        -0.021266481483774708,0.0,0.0,1.0,0.0,0.0,0.0,0.0,0.0,-0.0,-0.0,-1.0,-0.0,-0.0,-0.0,0.00058545213764139327,
        0.00069492775754933231,-0.013354826750081004,-0.015696387656065527,-0.016360391103343891,
        -0.0004481686028084641,0.013354826750081004,0.015696387656065527,0.016360391103343894,0.0,0.0,1.0,0.0,0.0,
        0.0,0.0,0.0,-0.0,-0.0,-1.0,-0.0,-0.0,-0.0,0.00070855886012245251,0.0163604987338591,-0.010053959431077385,
        -0.013815029502340643,-0.00070322802658466608,0.0,0.0,1.0,0.0,0.0,0.0,0.0,0.0,-0.0,-0.0,-1.0,-0.0,-0.0,-0.0,
        -0.0,0.00066290338327761684,0.00063267402481259919,-0.016360399418003064,0.013354829801521528,
        0.0156963952424949,0.016360399418003064,0.0,0.0,1.0,0.0,0.0,0.0,0.0,0.0,0.0,0.0,-0.0,-0.0,-1.0,-0.0,-0.0,
        -0.0,-0.0,0.00070871228093573281,-0.013354886628180915,-0.00070338839082327207,0.019136254043089867,
        0.019674776790317688,0.0,0.0,1.0,0.0,0.0,0.0,0.0,0.0,-0.0,-0.0,-1.0,-0.0,-0.0,-0.0,-0.0,-0.0,
        0.00070977892002071054,-0.015696489327294644,-0.00070486724956031889,0.0078498358546025652,
        0.021266597087506126,0.0,0.0,1.0,0.0,0.0,0.0,0.0,-0.0,-0.0,-1.0,-0.0,-0.0,-0.0,-0.0,0.00070855886012245251,
        -0.016360498733859103,-0.00070322802658466608,-0.00064115033886434007,0.010053959431077382,
        0.013815029502340643,0.0,0.0,1.0,0.0,0.0,0.0,0.0,-0.0,-0.0,-1.0,-0.0,-0.0,-0.0,-0.0,-0.0,
        0.015696429274739486,0.0007402725668637,0.013814978346247547,0.00078483961287594765,-0.0078505504957846264,
        -0.00059026517985183739,0.0,0.0,1.0,0.0,0.0,0.0,0.0,0.0,-0.0,-0.0,-1.0,-0.0,-0.0,-0.0,0.015696496781502492,
        0.00072094437214855291,0.013815028737181446,-0.0078505344125935073,-0.00078505003013483422,0.0,0.0,1.0,0.0,
        0.0,0.0,0.0,0.0,-0.0,-0.0,-1.0,-0.0,-0.0,-0.0,0.015696489327294647,0.00064281278721221359,
        0.013815029502340637,-0.0007099847981285385,-0.00785055587835492,0.00070514735512079252,0.0,0.0,1.0,0.0,0.0,
        0.0,0.0,0.0,-0.0,-0.0,-1.0,-0.0,-0.0,-0.0,-0.0,0.013814978346247547,-0.000740509959887708,
        -0.0078505513076336172,0.0005902592207076454,0.00045900348534280938,0.0,0.0,1.0,0.0,0.0,-0.0,-1.0,-0.0,-0.0,
        -0.0,0.00073887229766321256,0.016360436265260729,0.00078356528008410354,-0.00058935731463155463,
        -0.013814967279330388,0.0,0.0,1.0,0.0,0.0,0.0,0.0,0.0,-0.0,-0.0,-1.0,-0.0,-0.0,-0.0,0.00073903425520360994,
        0.019674701485866784,0.00078374994311404967,-0.01335483887448634,-0.00058948103625439357,
        0.019136152968431349,0.0,0.0,1.0,0.0,0.0,0.0,0.0,0.0,-0.0,-0.0,-1.0,-0.0,-0.0,-0.0,-0.0,
        0.0007402725668636999,0.00078483961287594722,-0.015696416044310803,-0.00059013581334217832,
        0.0078498304624371844,0.021266532224969138,0.0,0.0,0.0,0.0,0.0,-0.0,-1.0,-0.0,-0.0,-0.0,
        0.00073887229766321256,0.01005394241171902,0.01381497834624754,0.00078356528008410354,-0.016360422411734073,
        -0.00058935731463155463,0.0,0.0,1.0,0.0,0.0,0.0,0.0,-0.0,-0.0,-1.0,-0.0,-0.0,-0.0,-0.0,0.016360509090127547,
        0.00071950068311493818,-0.013815028737181451,-0.00078356528008410376,0.0,0.0,1.0,0.0,0.0,0.0,0.0,0.0,-0.0,
        -0.0,-1.0,-0.0,-0.0,-0.0,0.0163604987338591,-0.0007085588601224524,-0.013815029502340658,
        0.00070322802658466575,0.00064115033886434007,0.0,0.0,1.0,0.0,0.0,0.0,0.0,0.0,-0.0,-0.0,-1.0,-0.0,-0.0,-0.0,
        -0.0,0.016360436265260726,-0.00073887229766321266,-0.013814978346247555,0.00058935142225332476,
        0.00045695607481956147,0.0,0.0,1.0,0.0,0.0,-0.0,-1.0,-0.0,-0.0,-0.0,0.016360509090127547,
        -0.00071950068311493818,-0.010053942472644632,-0.013815028737181451,0.00066772991164514863,
        0.00078356528008410376,0.0,0.0,1.0,0.0,0.0,0.0,0.0,-0.0,-0.0,-1.0,-0.0,-0.0,-0.0,-0.0,
        0.00071965353685171413,-0.013354881724508197,-0.00078374994311405011,0.01913627908650653,
        0.019674802040209546,0.0,0.0,1.0,0.0,0.0,0.0,0.0,0.0,-0.0,-0.0,-1.0,-0.0,-0.0,-0.0,-0.0,
        0.00072094437214855281,-0.015696496781502488,-0.00078483961287594754,0.0078498143875897573,
        0.021266622548422189,0.0,0.0,0.0,0.0,0.0,-0.0,-1.0,-0.0,-0.0,-0.0,0.00071950068311493818,
        -0.016360509090127547,-0.00078356528008410376,0.010053942472644628,0.013815028737181455,0.0,0.0,1.0,0.0,0.0,
        0.0,0.0,-0.0,-0.0,-1.0,-0.0,-0.0,-0.0,-0.0,-0.013354886628180915,-0.00070871228093573313,
        0.019136254043089853,0.00070338839082327153,0.019674776790317681,0.00064128274259411333,0.0,0.0,1.0,0.0,0.0,
        0.0,0.0,0.0,-0.0,-0.0,-1.0,-0.0,-0.0,-0.0,-0.0,-0.0,-0.0078497740839998265,-0.01913681977138957,
        -0.00071047308705639756,0.021264803951796803,0.00072175936181417908,0.0,0.0,1.0,0.0,0.0,0.0,0.0,-0.0,-0.0,
        -1.0,-0.0,-0.0,-0.0,-0.0,-0.0,-0.013354847416887408,-0.00073903425520361,0.00058947514464916862,
        0.019136171450666897,0.019674701485866791,0.00045700543323026538,0.0,0.0,1.0,0.0,0.0,-0.0,-1.0,-0.0,-0.0,
        -0.0,-0.0,-0.010053984761327205,-0.019675305114254357,-0.0078504940691149945,-0.021264803951796817,
        -0.00071067908889347979,-0.00074130273940990277,-0.00072200639376403209,0.00071067908889347979,
        0.00072200639376403209,0.0,0.0,1.0,0.0,0.0,0.0,0.0,0.0,-0.0,-0.0,-1.0,-0.0,-0.0,-0.0,-0.0,-0.0,-0.0,
        -0.013354881724508197,-0.00071965353685171413,0.00066787723649602772,0.01913627908650652,
        0.00078374994311405,0.019674802040209542,0.0,0.0,1.0,0.0,0.0,0.0,0.0,-0.0,-0.0,-1.0,-0.0,-0.0,-0.0,-0.0,
        -0.0,-0.00070977892002071054,-0.015696489327294644,0.0078498358546025652,0.00070486724956031889,
        0.021266597087506126,0.00064281278721221337,0.0,0.0,0.0,0.0,0.0,-0.0,-1.0,-0.0,-0.0,-0.0,-0.0,
        -0.00058545213764139327,-0.00069492775754933231,-0.013354826750081004,-0.015696387656065527,
        -0.016360391103343891,0.013354826750081004,0.015696387656065527,0.016360391103343894,0.0004481686028084641,
        0.0,0.0,1.0,0.0,0.0,0.0,-0.0,-0.0,-1.0,-0.0,-0.0,-0.0,-0.0,-0.0,-0.00070855886012245251,
        -0.016360498733859103,0.010053959431077382,0.013815029502340643,0.00070322802658466608,
        0.00064115033886434007,0.0,0.0,1.0,0.0,0.0,0.0,0.0,-0.0,-0.0,-1.0,-0.0,-0.0,-0.0,-0.0,-0.0,
        -0.00066290338327761684,-0.00063267402481259919,-0.016360399418003064,0.013354829801521528,
        0.00082020698923774085,0.0,0.0,1.0,0.0,0.0,0.0,0.0,-0.0,-0.0,-1.0,-0.0,-0.0,-0.0,-0.0,-0.015696429274739486,
        -0.0007402725668637,0.0078498312759191675,0.0005901298647647122,0.021266544761989165,0.00045868723263609631,
        0.0,0.0,0.0,0.0,-1.0,-0.0,-0.0,-0.0,-0.015696496781502492,-0.013815028737181443,-0.00072119125834864851,
        0.0078505344125935142,0.00066885432718430675,0.00078505003013483422,0.0,0.0,1.0,0.0,0.0,0.0,-0.0,-0.0,-1.0,
        -0.0,-0.0,-0.0,-0.0,-0.0,-0.00073887229766321256,-0.016360436265260733,0.01005394241171902,
        0.00058935142225332476,0.013814978346247547,0.00045695607481956217,0.0,0.0,1.0,0.0,0.0,0.0,-0.0,-0.0,-1.0,
        -0.0,-0.0,-0.0,-0.0,-0.01636050909012755,-0.00071950068311493818,0.010053942472644628,
        0.00066772991164514863,0.01381502873718145,0.00078356528008410376,0.0,0.0,1.0,0.0,0.0,0.0,-0.0,-0.0,-1.0,
        -0.0,-0.0,-0.0,-0.0,-0.0,0.019136104037587275,0.0078505627081109745,0.00059070966910656456,
        4.6667541046249082E-6,-0.00046016924547736962,0.0,0.0,1.0,0.0,0.0,0.0,0.0,0.0,0.0,-0.0,-0.0,-1.0,-0.0,-0.0,
        -0.0,0.013354826750081004,0.000589475144649169,0.00070338839082327109,-0.019136104037587275,
        -0.00045721508909140403,0.0,0.0,1.0,0.0,0.0,0.0,-0.0,-1.0,-0.0,-0.0,-0.0,-0.0,0.01005395943107738,
        0.019674776790317691,0.0078505558783549187,0.00071067908889347968,-0.00070606688480528491,0.0,0.0,1.0,0.0,
        0.0,0.0,0.0,0.0,0.0,-0.0,-0.0,-1.0,-0.0,-0.0,-0.0,-0.0,0.01335483887448634,-0.00058948103625439325,-0.0,
        0.00045964338544026849,0.0078505504957846264,7.1576985742576626E-6,1.0242094517058181E-6,0.0,0.0,1.0,0.0,
        0.0,0.0,0.0,0.0,0.0,-0.0,-0.0,-1.0,-0.0,-0.0,-0.0,0.010053942472644626,0.019674802040209546,
        0.007850534412593509,0.021264422151952962,-0.00072200639376403209,0.00066940907433716364,
        0.00078577738649557045,0.0,0.0,1.0,0.0,0.0,0.0,0.0,0.0,-0.0,-0.0,-1.0,-0.0,-0.0,-0.0,-0.0,
        0.013354826750081004,-0.000589475144649169,-0.00070338839082327109,-0.019136104037587275,
        0.00045721508909140403,0.0,0.0,1.0,0.0,0.0,0.0,-0.0,-0.0,-1.0,-0.0,-0.0,-0.0,-0.0,-0.0,0.01335483887448634,
        -0.00078374994311405,-0.019136152968431349,-0.019674684401114268,0.00058948103625439325,0.0,0.0,1.0,0.0,0.0,
        0.0,0.0,-0.0,-0.0,-1.0,-0.0,-0.0,-0.0,-0.0,-0.0,0.00070998479812853861,0.013815029502340646,
        0.021266597087506119,-0.007850555878354917,-0.000705147355120792,0.0,0.0,1.0,0.0,0.0,0.0,0.0,0.0,-0.0,-0.0,
        -1.0,-0.0,-0.0,-0.0,-0.0,0.0007032280265846663,0.016360391103343884,0.000589357314631555,
        -0.013814936811065831,0.0,0.0,1.0,0.0,0.0,0.0,0.0,0.0,0.0,-0.0,-0.0,-1.0,-0.0,-0.0,-0.0,
        0.00058545773453366594,9.9821594966206443E-7,-0.013354818196216901,-0.015696374407663447,
        -0.016360377230620737,0.013354818196216901,0.015696374407663447,0.016360377230620737,0.0,0.0,1.0,0.0,0.0,
        0.0,0.0,0.0,0.0,0.0,-0.0,-0.0,-1.0,-0.0,-0.0,-0.0,-0.0,0.00070338839082327185,0.019674637958108528,
        0.00058948103625439336,-0.013354818196216903,0.019136085528464446,0.0,0.0,1.0,0.0,0.0,0.0,0.0,0.0,0.0,-0.0,
        -0.0,-1.0,-0.0,-0.0,-0.0,-0.0,0.0007048672495603191,0.00059013581334217821,-0.015696374407663444,
        0.00784984185776794,0.021266481483774712,0.0,0.0,0.0,0.0,0.0,0.0,-0.0,-1.0,-0.0,-0.0,-0.0,
        0.00058935142225332465,0.0007032280265846663,-0.016360391103343887,-0.0004571656718651675,
        0.010053943283910695,0.013814947892318402,0.0,0.0,1.0,0.0,0.0,0.0,0.0,-0.0,-0.0,-1.0,-0.0,-0.0,-0.0,
        0.00058935731463155485,1.0183040766464289E-6,-0.00013071479116047661,0.010053939720042822,
        0.013814936811065836,0.0,0.0,1.0,0.0,0.0,0.0,0.0,0.0,-0.0,-0.0,-1.0,-0.0,-0.0,-0.0,-0.0,
        0.00071047308705639756,-0.0078498358546025635,-0.019136254043089867,0.021264396690767625,0.0,0.0,1.0,0.0,
        0.0,0.0,0.0,-0.0,-0.0,-1.0,-0.0,-0.0,-0.0,-0.0,-0.0,0.00071029983670461863,0.00059047175686875969,
        -0.010053943283910698,-0.019674637958108521,-0.00045960759224737192,0.01804924706676608,0.0,1.0,0.0,0.0,0.0,
        0.0,-0.0,-0.0,-1.0,-0.0,-0.0,-0.0,-0.0,0.00070998479812853861,-0.013815029502340641,-0.000705147355120792,
        -0.00064310201354924451,0.007850555878354917,0.0,0.0,1.0,0.0,0.0,0.0,0.0,-0.0,-0.0,-1.0,-0.0,-0.0,-0.0,-0.0,
        -0.0,0.013815028737181446,0.021266622548422178,-0.00072119125834864851,-0.0078505344125935073,
        0.00066885432718430675,0.00078505003013483422,0.0,0.0,1.0,0.0,0.0,0.0,0.0,-0.0,-0.0,-1.0,-0.0,-0.0,-0.0,
        -0.0,0.013814947892318402,-0.0005902592207076454,-0.00070514735512079263,-0.0078505627081109815,
        0.00045921295820314543,0.0,0.0,1.0,0.0,0.0,-1.0,-0.0,-0.0,-0.0,-0.0,-0.0,0.015696416044310803,
        0.01381496727933039,-0.00078505003013483454,-0.0078505504957846247,0.00059026517985183728,0.0,0.0,1.0,0.0,
        0.0,0.0,0.0,-0.0,-0.0,-1.0,-0.0,-0.0,-0.0,-0.0,0.0007408652531395556,-0.010053942411719023,
        -0.019674701485866784,-0.00059047175686875969,-0.00045939812049741193,0.018049321508312247,0.0,1.0,0.0,0.0,
        0.0,-0.0,-0.0,-1.0,-0.0,-0.0,-0.0,-0.0,0.00074050995988770782,0.00078505003013483476,-0.013814967279330386,
        -0.00059026517985183717,0.007850550495784623,0.0,0.0,1.0,0.0,0.0,0.0,0.0,-0.0,-0.0,-1.0,-0.0,-0.0,-0.0,-0.0,
        0.016360391103343887,-0.00058935142225332465,-0.000703228026584666,-0.013814947892318404,
        0.00045716567186516885,0.0,0.0,1.0,0.0,0.0,-1.0,-0.0,-0.0,-0.0,-0.0,-0.0,-0.00066772991164514874,
        -0.00064115033886434018,-0.01381495313599773,0.00013071479116047655,-0.00058935731463155463,
        -0.010053939720042825,0.0,0.0,1.0,0.0,0.0,0.0,0.0,-0.0,-0.0,-1.0,-0.0,-0.0,-0.0,-0.0,-0.0,
        0.016360422411734077,-0.00078356528008410322,-0.010053938852608935,-0.013814967279330383,
        0.00058935731463155474,0.0,0.0,1.0,0.0,0.0,0.0,0.0,-0.0,-0.0,-1.0,-0.0,-0.0,-0.0,-0.0,
        0.00072155339410677672,-0.010053942472644626,-0.019674802040209542,-0.00078538438365502385,
        0.018049442230007151,0.0,0.0,1.0,0.0,0.0,0.0,0.0,-0.0,-0.0,-1.0,-0.0,-0.0,-0.0,-0.0,0.0007211912583486484,
        -0.01381502873718145,-0.00078505003013483443,0.0078505344125935073,0.0,0.0,1.0,0.0,0.0,0.0,0.0,-0.0,-0.0,
        -1.0,-0.0,-0.0,-0.0,-0.0,-0.010053959431077376,-0.00071029983670461863,-0.019674776790317688,
        -0.0078505558783549187,0.00070606688480528491,0.00064403085718071711,0.0,0.0,1.0,0.0,0.0,0.0,0.0,-0.0,-0.0,
        -1.0,-0.0,-0.0,-0.0,-0.0,-0.0,-0.0,-0.013354829801521528,-0.00066787723649602794,-0.00064128274259411312,
        0.019136117134310814,0.00082836908801823649,0.019674650101301497,0.0,1.0,0.0,0.0,0.0,0.0,-0.0,-0.0,-1.0,
        -0.0,-0.0,-0.0,-0.0,-0.0,-0.019136279086506527,-0.0078505344125935073,-0.018049442230007113,
        -0.00072200639376403209,0.00078577738649557045,0.0,0.0,1.0,0.0,0.0,0.0,-0.0,-0.0,-1.0,-0.0,-0.0,-0.0,-0.0,
        -0.0,-0.0,-0.010053942411719021,-0.0007408652531395556,-0.019674701485866787,0.00059047175686876,
        0.018049321508312247,0.00045939812049741166,0.0,1.0,0.0,0.0,-0.0,-1.0,-0.0,-0.0,-0.0,-0.0,
        -0.01335483887448634,-0.00078374994311405,0.00058948103625439325,0.019136152968431349,0.019674684401114268,
        0.0,0.0,1.0,0.0,0.0,0.0,0.0,-0.0,-0.0,-1.0,-0.0,-0.0,-0.0,-0.0,-0.0,-0.010053942472644626,
        -0.019674802040209546,-0.00072155339410677683,0.00066911306678242447,0.018049442230007123,
        0.00078538438365502352,0.0,1.0,0.0,0.0,0.0,-0.0,-0.0,-1.0,-0.0,-0.0,-0.0,-0.0,-0.00070998479812853861,
        -0.013815029502340641,0.007850555878354917,0.000705147355120792,0.00064310201354924451,0.0,0.0,1.0,0.0,0.0,
        0.0,0.0,-0.0,-0.0,-1.0,-0.0,-0.0,-0.0,-0.0,-0.0,-0.00066869452258176915,-0.015696395242494905,
        -0.00064281278721221348,0.0078498388863461367,0.00082974490333613884,0.021266503270189141,0.0,0.0,0.0,0.0,
        -0.0,-1.0,-0.0,-0.0,-0.0,-0.0,-0.00058545773453366594,-3.5950544673529394E-6,-0.013354818196216901,
        -0.015696374407663447,-0.016360377230620737,0.013354818196216901,0.015696374407663447,0.016360377230620737,
        0.0,0.0,1.0,0.0,0.0,0.0,0.0,0.0,-0.0,-0.0,-1.0,-0.0,-0.0,-0.0,-0.0,-0.0,-0.0,-0.013814978346247541,
        -0.00074050995988770782,0.0078505513076336225,0.00059025922070764572,0.00045900348534281133,0.0,0.0,1.0,0.0,
        0.0,0.0,-0.0,-0.0,-1.0,-0.0,-0.0,-0.0,-0.0,-0.015696416044310803,-0.00078483961287594765,
        0.0078498304624371948,0.00059013581334217821,0.021266532224969107,0.0,0.0,1.0,0.0,0.0,0.0,-0.0,-0.0,-1.0,
        -0.0,-0.0,-0.0,-0.0,-0.00078356528008410354,-0.016360422411734073,0.010053938852608933,
        0.00058935731463155463,0.013814967279330381,0.0,0.0,1.0,0.0,0.0,0.0,-0.0,-0.0,-1.0,-0.0,-0.0,-0.0,-0.0,-0.0,
        0.013354818196216903,0.00058948103625439347,0.0004572150890914036,-0.01913608552846445,0.0,0.0,1.0,0.0,0.0,
        0.0,0.0,0.0,0.0,-0.0,-0.0,-1.0,-0.0,-0.0,-0.0,-0.0,0.007850555878354917,4.72166684662135E-5,
        -0.00071067908889347968,0.00070606688480528491,0.00064403085718071711,0.0,0.0,1.0,0.0,0.0,0.0,0.0,0.0,0.0,
        -0.0,-0.0,-1.0,-0.0,-0.0,-0.0,-0.0,0.0078505513076336155,0.021264344306911508,-0.00074130273940990277,
        0.00059070966910656445,0.00045995981458200994,0.0,0.0,1.0,0.0,0.0,0.0,-0.0,-1.0,-0.0,-0.0,-0.0,
        0.019136104037587285,-0.00070578661505656148,0.0078505627081109728,-0.00059070966910656456,
        -4.6667541046249082E-6,0.00046016924547737027,0.0,0.0,1.0,0.0,0.0,-1.0,-0.0,-0.0,-0.0,-0.0,-0.0,
        0.010053938852608935,0.019674684401114268,-0.00078538438365502331,0.0078505504957846282,
        -7.1576985742576693E-6,0.00059071565881779026,0.0,0.0,1.0,0.0,0.0,0.0,0.0,0.0,-0.0,-0.0,-1.0,-0.0,-0.0,-0.0,
        -0.0,0.013354818196216903,-0.00058948103625439347,-0.00082836908801823736,-0.01913608552846445,
        -0.019674620847241392,0.0,0.0,1.0,0.0,0.0,0.0,0.0,-0.0,-0.0,-1.0,-0.0,-0.0,-0.0,-0.0,-0.0,-0.0,
        0.0078498304624371861,0.019136152968431349,-0.00078556684097776574,-0.021264331757721504,
        0.00059058621231803418,0.0,0.0,1.0,0.0,0.0,0.0,0.0,-0.0,-0.0,-1.0,-0.0,-0.0,-0.0,0.013814947892318409,
        0.0007051473551207923,0.0212664940442422,0.0005902651798518375,4.7206293852370952E-5,-0.007850561894963819,
        0.0,0.0,1.0,0.0,0.0,0.0,0.0,0.0,0.0,-0.0,-0.0,-1.0,-0.0,-0.0,-0.0,0.00059025922070764572,
        0.00070514735512079241,-0.013814947892318418,-0.00045921295820314608,0.0078505627081109711,0.0,0.0,1.0,0.0,
        0.0,0.0,0.0,-0.0,-0.0,-1.0,-0.0,-0.0,-0.0,1.0250173309722677E-6,0.0,-0.0,0.00059070966910656467,
        -0.0078505627081109745,-7.8752164488168983E-5,0.0,0.0,1.0,0.0,0.0,0.0,0.0,-0.0,-0.0,-1.0,-0.0,-0.0,-0.0,
        -0.0,0.00059026517985183772,1.0228783844071197E-6,-0.00012539822612430226,0.0078505618949638225,0.0,0.0,1.0,
        0.0,0.0,0.0,0.0,0.0,-0.0,-0.0,-1.0,-0.0,-0.0,-0.0,-0.0,0.00071067908889347979,-0.0078505558783549152,
        -7.8751758300344045E-5,-0.00070606688480528469,-0.00064403085718071711,0.0,0.0,1.0,0.0,0.0,0.0,0.0,-0.0,
        -0.0,-1.0,-0.0,-0.0,-0.0,-0.0,-0.0,-0.0,-0.00066885432718430643,-0.000643102013549245,-0.0078505589212312,
        0.00012539822612430221,-0.00059026517985183706,0.0,0.0,1.0,0.0,0.0,0.0,0.0,-0.0,-0.0,-1.0,-0.0,-0.0,-0.0,
        -0.0,-0.0,0.00045939812049741,-0.010053938852608933,-0.019674684401114268,-0.00059047772800183325,
        7.1576985742576753E-6,1.0242094517058098E-6,-0.00785055049578463,0.0,0.0,1.0,0.0,0.0,0.0,0.0,-0.0,-0.0,-1.0,
        -0.0,-0.0,-0.0,-0.0,-0.0,0.00074130273940990277,-0.00785055130763362,-0.018049321508312233,
        -0.00059070966910656445,-0.00045995981458201091,0.0,0.0,1.0,0.0,0.0,0.0,-0.0,-0.0,-1.0,-0.0,-0.0,-0.0,-0.0,
        -0.0,0.00072200639376403209,-0.007850534412593509,-0.018049442230007113,-0.00078577738649557056,0.0,0.0,1.0,
        0.0,0.0,0.0,0.0,-0.0,-0.0,-1.0,-0.0,-0.0,-0.0,-0.0,-0.0,-0.010053941700689279,-0.00066911306678242458,
        -0.019674650101301497,-0.00064350274257291972,0.018049261985986123,0.00083041340795978814,1.0,0.0,0.0,0.0,
        -0.0,-0.0,-1.0,-0.0,-0.0,-0.0,-0.0,-0.0,-0.013354818196216903,-0.00058948103625439347,
        -0.00082836908801823736,0.01913608552846445,0.019674620847241395,0.0,0.0,1.0,0.0,0.0,0.0,0.0,-0.0,-0.0,-1.0,
        -0.0,-0.0,-0.0,-0.0,-0.0,-0.0,-0.00074130273940990277,-0.0,-0.0078498304624371861,-0.019136152968431349,
        -0.00078556684097776574,0.00059058621231803418,0.0,0.0,1.0,0.0,0.0,0.0,-0.0,-0.0,-1.0,-0.0,-0.0,-0.0,-0.0,
        -0.0,-0.010053938852608928,-0.00078538438365502374,-0.019674684401114275,0.00059047772800183335,
        0.018049300450950378,0.0,1.0,0.0,0.0,0.0,-0.0,-0.0,-1.0,-0.0,-0.0,-0.0,-0.0,-0.015696374407663447,
        -0.0005902651798518375,-0.00012539822612430229,-1.0228783844071214E-6,0.007850561894963819,0.0,0.0,1.0,0.0,
        0.0,0.0,-0.0,-0.0,-1.0,-0.0,-0.0,-0.0,-0.0,-0.0,-0.0,-0.000589357314631555,-3.6300677219671527E-6,
        -0.00013071479116047663,0.01005393972004282,0.013814936811065819,0.0,0.0,1.0,0.0,0.0,0.0,-0.0,-0.0,-1.0,
        -0.0,-0.0,-0.0,-0.0,-0.0,-0.0,-0.013814967279330381,-0.00078505003013483476,-0.021266532224969107,
        -0.00045900348534281117,0.0078505504957846247,0.00059026517985183739,0.0,0.0,1.0,0.0,0.0,0.0,-0.0,-0.0,-1.0,
        -0.0,-0.0,-0.0,-0.0,-0.0,0.0078498418577679363,0.00059058621231803429,0.00012594643379194981,
        1.0243116170212105E-6,-0.021264280982048623,0.0,0.0,1.0,0.0,0.0,0.0,0.0,0.0,0.0,-0.0,-0.0,-1.0,-0.0,-0.0,
        -0.0,0.007850558921231196,-2.8452679316136533E-6,0.0008309073466565292,0.0,0.0,1.0,0.0,0.0,0.0,0.0,0.0,0.0,
        -0.0,-0.0,-1.0,-0.0,-0.0,-0.0,-0.0,0.0078498418577679328,-3.6410799041126835E-6,7.8752197135979057E-5,
        -0.00059071565881779048,-3.6422315821786528E-6,0.0,0.0,1.0,0.0,0.0,0.0,0.0,0.0,-0.0,-0.0,-1.0,-0.0,-0.0,
        -0.0,-0.0,-0.0,0.01005393972004282,8.6574413715050772E-5,-0.00059047772800183325,-0.018049225981178776,0.0,
        0.0,1.0,0.0,0.0,0.0,0.0,-0.0,-0.0,-1.0,-0.0,-0.0,-0.0,-0.0,-0.0,-0.01005393972004282,
        -0.00059047772800183325,-3.6400546269338619E-6,-8.6574413715050745E-5,0.018049225981178765,0.0,1.0,0.0,0.0,
        0.0,-0.0,-0.0,-1.0,-0.0,-0.0,-0.0,-0.0,-0.0,-0.0078498418577679363,-0.00012594643379194981,
        -0.00059071565881779048,-1.0250173309722696E-6,0.0,0.0,1.0,0.0,0.0,0.0,-0.0,-0.0,-1.0,-0.0,-0.0,-0.0,-0.0,
        -0.0,-0.0,-0.0,0.00785056189496382,0.00059071565881779048,4.721686715653703E-5,1.0250173309722696E-6,0.0,
        0.0,1.0,0.0,0.0,0.0,0.0,0.0,0.0,0.0,-0.0,-0.0,-1.0,-0.0,-0.0,-0.0,-0.002139599215214946,
        -0.023117048152407872,-0.0022397649528431126,-0.027072995129471072,-0.0021836277363616002,
        -0.028166145144496873,0.002139599215214946,0.023117048152407872,0.0022397649528431126,0.027072995129471072,
        0.0021836277363616007,0.028166145144496869,0.0,0.0,0.0,1.0,0.0,0.0,0.0,0.0,0.0,0.0,-0.0,-0.0,-0.0,-1.0,-0.0,
        -0.0,-0.0,-0.0,0.0021395992152149455,-0.023117145095115522,-0.0021497242199081533,-0.027072819798329567,
        -0.0019633569630565072,-0.02816590468451018,0.023117145095115522,0.027072819798329567,0.028165904684510173,
        0.0,0.0,0.0,1.0,0.0,0.0,0.0,0.0,0.0,-0.0,-0.0,-0.0,-1.0,-0.0,-0.0,-0.0,-0.0,0.023117048152407872,
        -0.0021505378228925251,-0.0022518711100377505,-0.032822477959688887,-0.00219585787232726,
        -0.0336642766045134,0.0021505378228925251,0.0022518711100377505,0.0021958578723272597,0.0,0.0,0.0,1.0,0.0,
        0.0,0.0,0.0,0.0,-0.0,-0.0,-0.0,-1.0,-0.0,-0.0,-0.0,-0.0,0.0022397649528431126,0.023117136629619534,
        0.028165879272568334,0.002368167038278622,-0.0017636731113387088,-0.023117134816530223,
        -0.027072790466377776,-0.028165871707620763,0.027072790466377776,0.0,0.0,0.0,1.0,0.0,0.0,0.0,0.0,0.0,-0.0,
        -0.0,-0.0,-1.0,-0.0,-0.0,-0.0,0.027072995129471072,0.0021528281310241241,0.0021984476162807444,
        0.023967033731365443,-0.0021532798422932995,-0.013757776970334581,-0.0022549381705200254,
        -0.002198962690806161,0.0,0.0,0.0,1.0,0.0,0.0,0.0,0.0,0.0,-0.0,-0.0,-0.0,-1.0,-0.0,-0.0,-0.0,
        0.0021836277363616002,-0.0020059903769841761,-0.023117107076915992,-0.0023681670382786246,
        -0.027072827080784432,-0.028165923858112191,0.023117107076915992,0.027072827080784432,0.028165923858112184,
        0.0,0.0,0.0,1.0,0.0,0.0,0.0,0.0,0.0,-0.0,-0.0,-0.0,-1.0,-0.0,-0.0,-0.0,0.028166145144496876,
        -0.0021508629271109274,-0.017539733206627071,-0.0022522704855525342,-0.023967033731365443,
        -0.0021962714305260589,0.0021508629271109274,0.0022522704855525342,0.0021962714305260593,0.0,0.0,0.0,1.0,
        0.0,0.0,0.0,0.0,0.0,-0.0,-0.0,-0.0,-1.0,-0.0,-0.0,-0.0,-0.0021395992152149455,-0.023117145095115522,
        -0.027072819798329567,-0.02816590468451018,0.023117145095115522,0.0021497242199081533,0.027072819798329567,
        0.0019633569630565077,0.028165904684510173,0.0,0.0,0.0,1.0,0.0,0.0,0.0,0.0,0.0,-0.0,-0.0,-0.0,-1.0,-0.0,
        -0.0,-0.0,-0.0,-0.023117048152407872,-0.0021505378228925251,-0.0022518711100377505,-0.00219585787232726,
        0.0021505378228925251,0.0022518711100377505,0.032822477959688887,0.0021958578723272597,0.033664276604513384,
        0.0,0.0,0.0,1.0,0.0,0.0,0.0,0.0,0.0,-0.0,-0.0,-0.0,-1.0,-0.0,-0.0,-0.0,-0.0,-0.0022397649528431126,
        -0.0023681670382786225,-0.023117134816530223,-0.027072790466377776,-0.028165871707620763,
        0.0017636731113387079,0.023117134816530223,0.028165871707620756,0.0,0.0,0.0,1.0,0.0,0.0,0.0,0.0,-0.0,-0.0,
        -0.0,-1.0,-0.0,-0.0,-0.0,-0.0,-0.027072995129471072,-0.0021528281310241241,-0.0021984476162807444,
        -0.023967033731365456,-0.0022549381705200254,0.0021532798422932995,0.013757776970334581,
        0.0022549381705200254,0.0021989626908061606,0.0,0.0,0.0,1.0,0.0,0.0,0.0,0.0,-0.0,-0.0,-0.0,-1.0,-0.0,-0.0,
        -0.0,-0.0,-0.0021836277363616007,-0.023117107076915992,-0.027072827080784432,-0.028165923858112191,
        0.0020059903769841761,0.023117107076915992,0.0023681670382786238,0.027072827080784432,0.028165923858112184,
        0.0,0.0,0.0,1.0,0.0,0.0,0.0,0.0,-0.0,-0.0,-0.0,-1.0,-0.0,-0.0,-0.0,-0.0,-0.028166145144496869,
        -0.0021508629271109274,-0.0022522704855525342,-0.0021962714305260589,0.0021508629271109274,
        0.017539733206627078,0.0022522704855525342,0.023967033731365467,0.0021962714305260593,0.0,0.0,0.0,1.0,0.0,
        0.0,0.0,0.0,-0.0,-0.0,-0.0,-1.0,-0.0,-0.0,-0.0,-0.0,0.0021505378228925246,0.023117145095115525,
        -0.0021629274560676956,-0.032821849572960068,-0.0019763195483343526,-0.033663644953626663,0.0,0.0,0.0,1.0,
        0.0,0.0,0.0,0.0,-0.0,-0.0,-0.0,-1.0,-0.0,-0.0,-0.0,-0.0,0.0021497242199081537,0.0017636731113387075,
        0.0025248548165844459,-0.023117153652107741,-0.027072767990336359,-0.028165839066171924,
        0.023117153652107741,0.027072767990336359,0.028165839066171917,0.0,0.0,0.0,1.0,0.0,0.0,0.0,0.0,0.0,0.0,-0.0,
        -0.0,-0.0,-1.0,-0.0,-0.0,-0.0,0.0021528281310241237,-0.013756932403821471,-0.03615897334115932,-0.0,
        0.0017730752489912573,0.027072767990336356,-0.036158836489428262,0.0,0.0,0.0,1.0,0.0,0.0,0.0,0.0,-0.0,-0.0,
        -0.0,-1.0,-0.0,-0.0,0.0020059903769841761,0.0019633569630565068,-0.023117148094275803,
        -0.0025248548165844454,0.028165850749951267,0.0,0.0,0.0,1.0,0.0,0.0,0.0,0.0,-0.0,-0.0,-0.0,-1.0,-0.0,-0.0,
        -0.0,0.0021508629271109274,-0.023967031267238804,-0.0,0.0017716448391260384,0.028165839066171927,0.0,0.0,
        0.0,1.0,0.0,0.0,0.0,0.0,0.0,-0.0,-0.0,-0.0,-1.0,-0.0,-0.0,0.0021505378228925246,-0.023117145095115525,-0.0,
        0.0017714658173675476,-0.0014235573934133095,0.033663511042732373,0.0,0.0,0.0,1.0,0.0,0.0,0.0,0.0,-0.0,-0.0,
        -0.0,-1.0,-0.0,-0.0,-0.0,0.0021528281310241237,-0.027072819798329564,-0.0021657727568646559,
        0.013756932403821471,0.036158973341159265,0.0,0.0,0.0,0.0,0.0,0.0,-0.0,-0.0,-0.0,-1.0,-0.0,-0.0,-0.0,
        0.0021508629271109274,-0.028165904684510176,-0.0021634485653239869,-0.0019768379174131762,
        0.017540054199611115,0.023967031267238814,0.0,0.0,0.0,1.0,0.0,0.0,0.0,-0.0,-0.0,-0.0,-1.0,-0.0,-0.0,-0.0,
        -0.0,0.023117136629619537,0.0022556280308783936,0.013758173064519321,-0.0017741542886565819,
        -0.0014273157197953927,0.0,0.0,0.0,1.0,0.0,0.0,0.0,0.0,-0.0,-0.0,-0.0,-1.0,-0.0,-0.0,0.013756545225322915,
        0.032822477959688887,-0.0021539160439461116,-0.002255628030878394,-0.0021996560033501643,
        -0.036155994182829158,0.0021539160439461116,0.002255628030878394,0.0021996560033501647,0.0,0.0,0.0,1.0,0.0,
        0.0,0.0,0.0,-0.0,-0.0,-0.0,-1.0,-0.0,-0.0,0.023117107076915996,0.0021958578723272597,-0.0020152870120824654,
        -0.0023798449910123255,-0.032821938754042893,0.0,0.0,0.0,1.0,0.0,0.0,0.0,0.0,-0.0,-0.0,-0.0,-1.0,-0.0,-0.0,
        -0.0,0.017539733206627082,0.0336642766045134,-0.00219941213896084,0.00215368729603372,0.0022553827543743792,
        0.00219941213896084,0.0,0.0,0.0,1.0,0.0,0.0,0.0,0.0,0.0,0.0,-0.0,-0.0,-0.0,-1.0,-0.0,-0.0,-0.0,
        0.023117145095115518,-0.0021505378228925251,-0.032821849572960082,0.0021629274560676964,
        0.0019763195483343534,0.0,0.0,0.0,1.0,0.0,0.0,0.0,0.0,-0.0,-0.0,-0.0,-1.0,-0.0,-0.0,-0.0,-0.0,
        0.023117136629619537,-0.00225187111003775,-0.032821807333186945,0.0017714658173675487,0.0014229487589399608,
        0.0,0.0,0.0,1.0,0.0,0.0,0.0,-0.0,-0.0,-0.0,-1.0,-0.0,-0.0,-0.0,0.023117107076915996,-0.0021958578723272597,
        -0.032821938754042893,-0.033663737674327086,0.0020152870120824654,0.0023798449910123263,0.0,0.0,0.0,1.0,0.0,
        0.0,0.0,-0.0,-0.0,-0.0,-1.0,-0.0,-0.0,-0.0,-0.0,0.0022544308843389775,0.027072797014430487,
        0.0023823041653880553,0.023967015852373385,-0.0017733843081747245,-0.013758177150392206,0.0,0.0,0.0,1.0,0.0,
        0.0,0.0,0.0,-0.0,-0.0,-0.0,-1.0,-0.0,-0.0,0.0022522704855525342,0.028165879272568337,0.0023802034757232954,
        -0.0017716448391260397,-0.023967012140249259,0.0,0.0,0.0,1.0,0.0,0.0,0.0,0.0,-0.0,-0.0,-0.0,-1.0,-0.0,-0.0,
        0.0022518711100377505,0.03366360485977575,0.0023798449910123263,-0.023117134816530216,
        -0.0017714855698833817,0.032821793825602318,0.0,0.0,0.0,1.0,0.0,0.0,0.0,0.0,-0.0,-0.0,-0.0,-1.0,-0.0,-0.0,
        -0.0,0.0023823041653880553,-0.027072790466377783,-0.0017730752489912573,0.01375694528625826,
        0.036158931786919049,0.0,0.0,0.0,0.0,0.0,-0.0,-0.0,-1.0,-0.0,-0.0,0.027072827080784432,
        0.0021984476162807444,0.023967007687598831,-0.013758082261467377,-0.0023827866608640042,0.0,0.0,0.0,1.0,0.0,
        0.0,0.0,0.0,-0.0,-0.0,-0.0,-1.0,-0.0,-0.0,0.027072819798329564,0.0019791101348432538,0.0239670312672388,
        -0.0021532798422932995,-0.013758164253474777,0.0021663421034936255,0.0,0.0,0.0,1.0,0.0,0.0,0.0,0.0,-0.0,
        -0.0,-0.0,-1.0,-0.0,-0.0,-0.0,0.02707279701443048,0.023967015852373378,-0.0022549381705200249,
        -0.013758173064519324,0.0017733644650094233,0.001426115796022355,0.0,0.0,1.0,0.0,0.0,-0.0,-0.0,-1.0,-0.0,
        -0.0,0.027072827080784432,0.0020172069825707454,0.0023823041653880544,0.023967007687598831,
        -0.00219896269080616,-0.013758082261467377,0.0,0.0,0.0,1.0,0.0,0.0,0.0,-0.0,-0.0,-0.0,-1.0,-0.0,-0.0,-0.0,
        0.0021962714305260589,0.028165923858112184,-0.0023802034757232967,-0.023967007687598837,0.0,0.0,0.0,1.0,0.0,
        0.0,0.0,0.0,-0.0,-0.0,-0.0,-1.0,-0.0,-0.0,0.0021958578723272597,-0.023117107076915992,
        -0.0023798449910123281,0.032821938754042886,0.033663737674327066,0.0,0.0,0.0,1.0,0.0,0.0,0.0,0.0,-0.0,-0.0,
        -0.0,-1.0,-0.0,-0.0,-0.0,0.002198447616280744,-0.027072827080784435,-0.0023823041653880561,
        0.013756850421972387,0.036159076531973151,0.0,0.0,0.0,0.0,0.0,-0.0,-0.0,-1.0,-0.0,-0.0,
        0.0021962714305260589,-0.028165923858112181,-0.0020155176559669297,-0.0023802034757232967,
        0.017539980122310408,0.023967007687598862,0.0,0.0,0.0,1.0,0.0,0.0,0.0,-0.0,-0.0,-0.0,-1.0,-0.0,-0.0,-0.0,
        0.02816590468451018,-0.0021508629271109274,-0.023967031267238807,0.0021634485653239869,
        0.0019768379174131758,0.0,0.0,0.0,1.0,0.0,0.0,0.0,0.0,-0.0,-0.0,-0.0,-1.0,-0.0,-0.0,-0.0,
        0.028165879272568337,-0.0022522704855525342,-0.023967015852373392,0.0017716250685312594,
        0.0014234593859236441,0.0,0.0,1.0,0.0,0.0,-0.0,-0.0,-1.0,-0.0,-0.0,0.028165923858112191,
        -0.0021962714305260589,-0.023967007687598817,0.0020155176559669297,0.0023802034757232963,0.0,0.0,0.0,1.0,
        0.0,0.0,0.0,-0.0,-0.0,-0.0,-1.0,-0.0,-0.0,-0.0,-0.0021505378228925246,-0.023117145095115525,
        0.0021629274560676956,0.032821849572960068,0.001976319548334353,0.033663644953626656,0.0,0.0,0.0,1.0,0.0,
        0.0,0.0,0.0,-0.0,-0.0,-0.0,-1.0,-0.0,-0.0,-0.0,-0.0,-0.0017636536977724872,-0.0021497242199081537,
        -0.023117155475339022,0.0014113188375514472,0.028165846654428471,0.0,0.0,0.0,1.0,0.0,0.0,0.0,-0.0,-0.0,-0.0,
        -1.0,-0.0,-0.0,-0.0,-0.0,-0.0021528281310241237,-0.027072819798329564,0.013756932403821471,
        0.0021657727568646559,0.0019791101348432556,0.036158973341159265,0.0,0.0,0.0,0.0,0.0,-0.0,-0.0,-1.0,-0.0,
        -0.0,-0.0,-0.0020059903769841757,-0.0019633569630565077,-0.0017636731113387079,-0.0014113188375514463,
        -0.023117153652107741,-0.027072767990336359,-0.028165839066171924,0.023117153652107741,0.028165839066171917,
        0.0,0.0,0.0,1.0,0.0,0.0,0.0,0.0,-0.0,-0.0,-0.0,-1.0,-0.0,-0.0,-0.0,-0.0,-0.0,-0.0021508629271109274,
        -0.028165904684510176,0.017540054199611115,0.0021634485653239869,0.023967031267238814,0.0019768379174131762,
        0.0,0.0,0.0,1.0,0.0,0.0,0.0,-0.0,-0.0,-0.0,-1.0,-0.0,-0.0,-0.0,-0.0,-0.023117136629619537,
        -0.00225187111003775,0.0017714658173675487,0.032821807333186945,0.0014229487589399608,0.033663604859775743,
        0.0,0.0,1.0,0.0,0.0,-0.0,-0.0,-1.0,-0.0,-0.0,-0.0,-0.013756545225322915,-0.032822477959688887,
        -0.0021539160439461116,-0.002255628030878394,-0.0021996560033501643,0.0021539160439461116,
        0.002255628030878394,0.0021996560033501647,0.036155994182829096,0.0,0.0,0.0,0.0,0.0,0.0,-0.0,-0.0,-0.0,-1.0,
        -0.0,-0.0,-0.0,-0.0,-0.023117107076915996,-0.0021958578723272597,0.0020152870120824654,
        0.0023798449910123263,0.032821938754042893,0.033663737674327072,0.0,0.0,0.0,1.0,0.0,0.0,0.0,-0.0,-0.0,-0.0,
        -1.0,-0.0,-0.0,-0.0,-0.0,-0.017539733206627085,-0.033664276604513384,-0.00219941213896084,
        0.00215368729603372,0.03112680478206669,0.0,0.0,0.0,1.0,0.0,0.0,0.0,-0.0,-0.0,-0.0,-1.0,-0.0,-0.0,-0.0,
        -0.0022544308843389775,-0.027072797014430487,0.0017730554216371041,0.013756941202814331,
        0.0014255752842010033,0.0361589433554084,0.0,0.0,0.0,0.0,-0.0,-1.0,-0.0,-0.0,-0.0022522704855525342,
        -0.0023802034757232954,-0.028165871707620752,0.00177164483912604,0.017540060210790732,0.023967012140249284,
        0.0,0.0,0.0,1.0,0.0,0.0,-0.0,-0.0,-0.0,-1.0,-0.0,-0.0,-0.0,-0.0,-0.027072827080784432,
        -0.0021984476162807448,0.0020172069825707454,0.013756850421972387,0.0023823041653880557,
        0.036159076531973207,0.0,0.0,0.0,1.0,0.0,0.0,-0.0,-0.0,-0.0,-1.0,-0.0,-0.0,-0.0,-0.0021962714305260593,
        -0.028165923858112181,0.0020155176559669297,0.017539980122310408,0.0023802034757232963,0.023967007687598862,
        0.0,0.0,0.0,1.0,0.0,0.0,-0.0,-0.0,-0.0,-1.0,-0.0,-0.0,-0.0,-0.0,0.0021670637484648039,0.0017738649457463914,
        0.013757007748269136,0.00021693526799154337,-0.036155235792572543,0.0,0.0,0.0,1.0,0.0,0.0,0.0,0.0,0.0,-0.0,
        -0.0,-0.0,-1.0,-0.0,-0.0,0.002153916043946112,0.013756932403821469,0.032821849572960068,
        -0.002167063748464803,-0.036155372747005976,0.0,0.0,0.0,1.0,0.0,0.0,-0.0,-0.0,-1.0,-0.0,-0.0,-0.0,
        0.002015287012082465,0.0019763195483343526,0.0017714855698833811,0.023117153652107737,-0.032821701216996041,
        0.0,0.0,0.0,1.0,0.0,0.0,0.0,0.0,0.0,-0.0,-0.0,-0.0,-1.0,-0.0,-0.0,-0.0,0.002153279842293299,
        -0.013758164253474777,-0.0,0.036158848104067796,0.0017733843081747236,0.00021831715113692992,
        8.0516212332184942E-5,0.0,0.0,0.0,1.0,0.0,0.0,0.0,0.0,0.0,-0.0,-0.0,-0.0,-1.0,-0.0,-0.0,
        0.0020155176559669297,0.0019768379174131766,0.0017716448391260384,0.0014240679527817289,
        -0.02816583906617192,0.017540113132327881,0.023967016586099663,0.0,0.0,0.0,1.0,0.0,0.0,0.0,0.0,-0.0,-0.0,
        -0.0,-1.0,-0.0,-0.0,-0.0,0.002153916043946112,-0.013756932403821469,-0.032821849572960068,
        -0.002167063748464803,0.036155372747005914,0.0,0.0,0.0,0.0,0.0,0.0,-0.0,-0.0,-0.0,-1.0,-0.0,-0.0,-0.0,-0.0,
        0.002153279842293299,-0.023967031267238814,-0.0021663421034936268,-0.0019796723009276795,
        0.013758164253474772,0.0,0.0,0.0,1.0,0.0,0.0,0.0,-0.0,-0.0,-0.0,-1.0,-0.0,-0.0,-0.0,-0.0,
        0.023117134816530216,0.0023798449910123268,0.0014229487589399567,-0.001771485569883382,
        -0.032821793825602304,0.0,0.0,0.0,1.0,0.0,0.0,0.0,0.0,-0.0,-0.0,-0.0,-1.0,-0.0,-0.0,-0.0,
        0.032821938754042893,0.0021996560033501643,0.013758082261467375,-0.00238394443966586,0.0,0.0,0.0,1.0,0.0,
        0.0,0.0,0.0,0.0,-0.0,-0.0,-0.0,-1.0,-0.0,-0.0,0.013757776970334586,8.0531054257304872E-5,
        -0.0021543679790237634,-0.0022561355647809592,-0.002200171328627197,0.0021543679790237634,
        0.0022561355647809592,0.002200171328627197,0.0,0.0,0.0,1.0,0.0,0.0,0.0,0.0,0.0,0.0,-0.0,-0.0,-0.0,-1.0,-0.0,
        -0.0,-0.0,0.032821849572960062,0.0019803784157214573,0.013758164253474772,-0.0021543679790237639,
        0.0021676333667632283,0.0,0.0,0.0,1.0,0.0,0.0,0.0,0.0,0.0,-0.0,-0.0,-0.0,-1.0,-0.0,-0.0,-0.0,
        0.032821807333186952,0.013758173064519319,-0.0022561355647809588,0.0017741542886565826,
        0.0014273157197953908,0.0,0.0,1.0,0.0,0.0,0.0,-0.0,-0.0,-1.0,-0.0,-0.0,0.013756850421972394,
        0.032821938754042893,-0.0021996560033501647,-0.036155475949002973,0.0020181389031338108,
        0.0023834617064148775,0.0,0.0,0.0,1.0,0.0,0.0,0.0,-0.0,-0.0,-0.0,-1.0,-0.0,-0.0,0.013758082261467373,
        8.05337557427544E-5,-1.7578747218645929E-5,0.0020185138829726234,0.0023839444396658582,0.0,0.0,0.0,1.0,0.0,
        0.0,0.0,0.0,-0.0,-0.0,-0.0,-1.0,-0.0,-0.0,-0.0,0.023117155475339025,-0.0017714658173675481,
        -0.0021629274560676964,0.0014235573934133154,0.0,0.0,0.0,1.0,0.0,0.0,0.0,-0.0,-0.0,-0.0,-1.0,-0.0,-0.0,-0.0,
        -0.0,0.023117148094275806,0.013756987718843332,-0.0020181389031338121,-0.0019803784157214573,
        -0.036155266228744543,0.0025428266645309921,0.0,0.0,1.0,0.0,0.0,0.0,-0.0,-0.0,-0.0,-1.0,-0.0,-0.0,-0.0,
        0.023117134816530216,-0.0023798449910123259,-0.032821793825602304,-0.033663591643505526,
        0.0017714855698833828,0.0,0.0,0.0,1.0,0.0,0.0,0.0,-0.0,-0.0,-0.0,-1.0,-0.0,-0.0,-0.0,-0.0,
        0.0023802034757232954,0.0014234593859236444,-0.028165871707620752,-0.0017716448391260397,
        0.017540060210790732,0.023967012140249284,0.0,0.0,0.0,1.0,0.0,0.0,0.0,-0.0,-0.0,-0.0,-1.0,-0.0,-0.0,-0.0,
        0.0023834617064148788,-0.01375694528625827,-0.032821793825602311,-0.0017738649457463916,0.03615533112817032,
        0.0,0.0,0.0,0.0,0.0,-0.0,-1.0,-0.0,-0.0,-0.0,-0.0,0.0022549381705200249,0.0023827866608640046,
        -0.02396701214024928,-0.0017733843081747234,0.0137581771503922,0.0,0.0,0.0,1.0,0.0,0.0,0.0,-0.0,-0.0,-0.0,
        -1.0,-0.0,-0.0,-0.0,0.027072776376697909,-0.0020172069825707458,-0.0019791101348432543,
        -0.013756987718843334,-0.036158866905630971,0.0025414906519322343,0.0,0.0,1.0,0.0,0.0,-0.0,-0.0,-0.0,-1.0,
        -0.0,-0.0,-0.0,0.027072790466377776,0.023967012140249266,-0.0023827866608640033,-0.013758177150392204,
        0.0017733843081747238,0.0,0.0,0.0,1.0,0.0,0.0,0.0,-0.0,-0.0,-0.0,-1.0,-0.0,-0.0,-0.0,0.0021996560033501638,
        -0.013756850421972376,-0.032821938754042906,-0.0023834617064148788,0.036155475949002897,0.0,0.0,0.0,0.0,0.0,
        -0.0,-1.0,-0.0,-0.0,-0.0,-0.0,-0.0175399801223104,-0.033663737674327059,-0.0023832147743805109,
        1.7578747218645923E-5,-0.013758082261467368,-0.002018513882972623,0.0,0.0,0.0,1.0,0.0,0.0,0.0,-0.0,-0.0,
        -0.0,-1.0,-0.0,-0.0,-0.0,-0.0,0.00219896269080616,-0.023967007687598848,-0.0020175817725937989,
        -0.0023827866608640037,0.013758082261467373,0.0,0.0,0.0,1.0,0.0,0.0,0.0,-0.0,-0.0,-0.0,-1.0,-0.0,-0.0,-0.0,
        0.02816585074995127,-0.0020155176559669297,-0.0019768379174131762,-0.023967016242290962,
        0.0025390630631617036,0.0,0.0,0.0,1.0,0.0,0.0,0.0,-0.0,-0.0,-0.0,-1.0,-0.0,-0.0,-0.0,0.028165871707620759,
        -0.0023802034757232963,-0.023967012140249263,0.0017716448391260375,0.0,0.0,0.0,1.0,0.0,0.0,0.0,-0.0,-0.0,
        -0.0,-1.0,-0.0,-0.0,-0.0,-0.002015287012082465,-0.023117148094275806,-0.0019763195483343526,
        -0.0017714855698833811,0.032821701216996041,0.0336634977860711,0.0,0.0,0.0,1.0,0.0,0.0,0.0,-0.0,-0.0,-0.0,
        -1.0,-0.0,-0.0,-0.0,-0.0,-0.0,-0.0021536872960337197,-0.017540054199611122,-0.033663644953626642,
        0.0021668136920060164,0.03112619259567026,0.0019801394547201774,0.0,0.0,1.0,0.0,0.0,0.0,-0.0,-0.0,-0.0,-1.0,
        -0.0,-0.0,-0.0,-0.0,-0.0021634485653239878,-0.0017716448391260386,-0.0025390630631616988,
        -0.02816583906617192,0.023967016586099663,0.0,0.0,0.0,1.0,0.0,0.0,-0.0,-0.0,-0.0,-1.0,-0.0,-0.0,-0.0,-0.0,
        -0.0,-0.0020172069825707454,-0.027072776376697909,-0.0019791101348432543,0.013756987718843336,
        0.0025414906519322382,0.036158866905630881,0.0,0.0,0.0,0.0,-0.0,-0.0,-1.0,-0.0,-0.0,-0.0,
        -0.002153279842293299,-0.023967031267238814,0.013758164253474772,0.0021663421034936268,0.00197967230092768,
        0.0,0.0,0.0,1.0,0.0,0.0,0.0,-0.0,-0.0,-0.0,-1.0,-0.0,-0.0,-0.0,-0.0,-0.0020155176559669297,
        -0.0019768379174131771,-0.02816585074995127,0.017540096325751132,0.0025390630631616997,0.023967016242290966,
        0.0,0.0,1.0,0.0,0.0,-0.0,-0.0,-0.0,-1.0,-0.0,-0.0,-0.0,-0.023117134816530216,-0.0023798449910123259,
        0.0017714855698833828,0.032821793825602304,0.033663591643505512,0.0,0.0,0.0,1.0,0.0,0.0,0.0,-0.0,-0.0,-0.0,
        -1.0,-0.0,-0.0,-0.0,-0.0,-0.017540057790927686,-0.0022553827543743796,-0.033663604859775743,
        0.0017736671849664688,0.031126147710011594,0.00142656920316686,0.0,1.0,0.0,0.0,-0.0,-0.0,-1.0,-0.0,-0.0,
        -0.0,-0.013757776970334586,-0.00013643209586666446,-0.0021543679790237634,-0.0022561355647809592,
        -0.002200171328627197,0.0021543679790237634,0.0022561355647809592,0.002200171328627197,0.0,0.0,0.0,1.0,0.0,
        0.0,0.0,0.0,-0.0,-0.0,-0.0,-1.0,-0.0,-0.0,-0.0,-0.0,-0.0,-0.0023823041653880544,-0.027072790466377773,
        0.0017730752489912573,0.013756945286258279,0.036158931786919229,0.0,0.0,0.0,1.0,0.0,0.0,-0.0,-0.0,-0.0,-1.0,
        -0.0,-0.0,-0.0,-0.0022549381705200249,-0.0239670158523734,0.0017733644650094235,0.013758173064519321,
        0.0014261157960223586,0.0,0.0,0.0,1.0,0.0,0.0,-0.0,-0.0,-0.0,-1.0,-0.0,-0.0,-0.0,-0.023967007687598844,
        -0.00219896269080616,0.0020175817725937989,0.013758082261467377,0.0023827866608640033,0.0,0.0,0.0,1.0,0.0,
        0.0,-0.0,-0.0,-0.0,-1.0,-0.0,-0.0,-0.0,-0.0,0.0021543679790237634,0.013758164253474772,0.03615537274700599,
        -0.0021676333667632296,0.0,0.0,0.0,1.0,0.0,0.0,0.0,0.0,0.0,-0.0,-0.0,-0.0,-1.0,-0.0,-0.0,-0.0,
        0.001771485569883382,3.1609473085406838E-6,-0.023117153652107744,0.032821701216996027,0.033663497786071091,
        0.0,0.0,0.0,1.0,0.0,0.0,0.0,0.0,0.0,-0.0,-0.0,-0.0,-1.0,-0.0,-0.0,-0.0,0.0017730752489912571,
        0.0014261840281970283,-0.027072767990336359,0.013757007748269138,0.036158836489428171,0.0,0.0,0.0,0.0,0.0,
        0.0,-0.0,-0.0,-1.0,-0.0,-0.0,0.0021670637484648039,-0.032821714763063607,0.0017738649457463914,
        -0.013757007748269151,-0.00021693526799154326,0.036155235792572536,0.0,0.0,0.0,0.0,0.0,-0.0,-1.0,-0.0,-0.0,
        -0.0,-0.0,0.0020175817725937989,0.0019796723009276795,-0.023967016242290948,0.001773384308174724,
        -0.00021831715113693025,0.013758239625790694,0.0,0.0,0.0,1.0,0.0,0.0,0.0,0.0,-0.0,-0.0,-0.0,-1.0,-0.0,-0.0,
        -0.0,0.0021543679790237634,-0.013758164253474772,-0.031126192595670284,-0.0021676333667632296,
        -0.0019809408498811915,0.0,0.0,0.0,1.0,0.0,0.0,0.0,-0.0,-0.0,-0.0,-1.0,-0.0,-0.0,-0.0,-0.0,-0.0,
        0.0017733644650094228,0.0021663421034936259,-0.02396702031125434,-0.0014267245515185119,
        0.013758235536900225,0.0,0.0,0.0,1.0,0.0,0.0,0.0,-0.0,-0.0,-0.0,-1.0,-0.0,-0.0,0.0023834617064148775,
        0.032821793825602311,0.0014267749509501136,0.013758177150392209,3.1682855172904752E-6,
        -0.0017741741644841874,0.0,0.0,0.0,1.0,0.0,0.0,0.0,0.0,0.0,-0.0,-0.0,-0.0,-1.0,-0.0,-0.0,
        0.013756945286258268,0.032821793825602311,-0.002383461706414877,-0.036155331128170466,0.0017738649457463927,
        0.0,0.0,0.0,1.0,0.0,0.0,0.0,-0.0,-0.0,-0.0,-1.0,-0.0,-0.0,8.0535028485727747E-5,0.0,-0.0,
        0.013757007748269136,-0.0017738649457463922,-1.1094817584871507E-5,0.0,0.0,0.0,1.0,0.0,0.0,0.0,-0.0,-0.0,
        -0.0,-1.0,-0.0,-0.0,-0.0,0.013758177150392211,8.05345450981963E-5,-2.1639071390723852E-5,
        0.0017741741644841872,0.0,0.0,0.0,1.0,0.0,0.0,0.0,0.0,-0.0,-0.0,-0.0,-1.0,-0.0,-0.0,-0.0,
        0.023117153652107741,-0.0017714855698833822,-1.107593583908204E-5,-0.032821701216996048,
        -0.033663497786071112,0.0,0.0,0.0,1.0,0.0,0.0,0.0,-0.0,-0.0,-0.0,-1.0,-0.0,-0.0,-0.0,-0.0,-0.0,
        -0.017540060210790728,-0.033663591643505519,-0.001773687040351414,2.1639071390723859E-5,
        -0.013758177150392211,0.0,0.0,0.0,1.0,0.0,0.0,0.0,-0.0,-0.0,-0.0,-1.0,-0.0,-0.0,-0.0,-0.0,
        0.036158866905630936,-0.0020175817725937989,-0.0019796723009276795,-0.013758219590295969,
        0.00021831715113693025,8.0516212332184712E-5,-0.0017733843081747243,0.0,0.0,0.0,1.0,0.0,0.0,0.0,-0.0,-0.0,
        -0.0,-1.0,-0.0,-0.0,-0.0,-0.0,0.027072767990336359,-0.0017730752489912582,-0.0025414906519322356,
        -0.013757007748269127,-0.036158836489428296,0.0,0.0,0.0,1.0,0.0,0.0,-0.0,-0.0,-0.0,-1.0,-0.0,-0.0,-0.0,-0.0,
        0.02816583906617192,-0.0017716448391260386,-0.0025390630631616979,-0.023967016586099656,0.0,0.0,0.0,1.0,0.0,
        0.0,0.0,-0.0,-0.0,-0.0,-1.0,-0.0,-0.0,-0.0,-0.0,-0.002017933713019439,-0.017540096325751129,
        -0.0019801394547201766,-0.033663529390784139,0.0025425544502436937,0.031126075963179154,0.0,1.0,0.0,0.0,
        -0.0,-0.0,-0.0,-1.0,-0.0,-0.0,-0.0,-0.0,-0.0021543679790237634,-0.013758164253474772,-0.031126192595670284,
        0.0021676333667632296,0.0019809408498811919,0.0,0.0,0.0,1.0,0.0,0.0,0.0,-0.0,-0.0,-0.0,-1.0,-0.0,-0.0,-0.0,
        -0.0,-0.0,-0.027072767990336356,-0.0,-0.0017733644650094228,-0.0021663421034936259,-0.02396702031125434,
        0.013758235536900225,0.0,0.0,0.0,1.0,0.0,0.0,-0.0,-0.0,-0.0,-1.0,-0.0,-0.0,-0.0,-0.0,-0.0020175817725937989,
        -0.023967016242290959,-0.00197967230092768,0.013758219590295984,0.0025420742486267352,0.0,0.0,1.0,0.0,0.0,
        -0.0,-0.0,-0.0,-1.0,-0.0,-0.0,-0.0,-0.0022561355647809592,-0.013758177150392209,-2.1639071390723856E-5,
        -8.0534545098196153E-5,0.0017741741644841874,0.0,0.0,0.0,1.0,0.0,0.0,-0.0,-0.0,-0.0,-1.0,-0.0,-0.0,-0.0,
        -0.0,-0.0,-0.013758082261467375,-0.00013643680450863756,-1.7578747218645926E-5,0.0020185138829726234,
        0.0023839444396658587,0.0,0.0,0.0,1.0,0.0,0.0,-0.0,-0.0,-0.0,-1.0,-0.0,-0.0,-0.0,-0.0,-0.0,
        -0.0023827866608640033,-0.023967012140249294,-0.001426115796022355,-0.036158931786919105,
        0.0017733843081747249,0.013758177150392206,0.0,0.0,0.0,1.0,0.0,0.0,-0.0,-0.0,-0.0,-1.0,-0.0,-0.0,-0.0,-0.0,
        0.0017741542886565815,0.013758235536900216,1.4266538049601484E-5,8.0534981096103676E-5,
        -0.0014279245624933968,0.0,0.0,0.0,1.0,0.0,0.0,0.0,0.0,0.0,-0.0,-0.0,-0.0,-1.0,-0.0,-0.0,
        0.0017736870403514127,-0.00014872217635028418,0.031126045000755019,0.0,0.0,0.0,0.0,0.0,0.0,0.0,0.0,0.0,-0.0,
        -0.0,-0.0,-1.0,-0.0,-0.0,-0.0,0.0017741542886565813,-0.00013643903899346717,1.1097382704726312E-5,
        -0.01375823962579072,-0.00013643911633017095,0.0,0.0,0.0,1.0,0.0,0.0,0.0,0.0,-0.0,-0.0,-0.0,-1.0,-0.0,-0.0,
        -0.0,-0.0,0.0020185138829726234,8.7167521048673558E-6,-0.013758219590295984,-0.0025434105399164903,0.0,0.0,
        0.0,1.0,0.0,0.0,0.0,-0.0,-0.0,-0.0,-1.0,-0.0,-0.0,-0.0,-0.0,-0.0020185138829726234,-0.013758219590295977,
        -0.00013643880956405708,-8.7167521048673558E-6,0.0025434105399164829,0.0,0.0,1.0,0.0,0.0,-0.0,-0.0,-0.0,
        -1.0,-0.0,-0.0,-0.0,-0.0,-0.0017741542886565815,-1.4266538049601484E-5,-0.013758239625790697,
        -8.0535028485727734E-5,0.0,0.0,0.0,1.0,0.0,0.0,-0.0,-0.0,-0.0,-1.0,-0.0,-0.0,-0.0,-0.0,-0.0,-0.0,
        0.0017741741644841864,0.013758239625790697,3.1706750128877981E-6,8.0535028485727883E-5,0.0,0.0,0.0,1.0,0.0,
        0.0,0.0,0.0,0.0,0.0,-0.0,-0.0,-0.0,-1.0,-0.0,-0.0,-0.555673663731469,-0.026771909379554294,
        -0.62490021645747618,-0.027265477962947069,-0.63800507768378811,-0.026352061912650541,0.555673663731469,
        0.026771909379554294,0.62490021645747618,0.027265477962947066,0.63800507768378822,0.026352061912650541,0.0,
        0.0,0.0,0.0,1.0,0.0,0.0,0.0,0.0,0.0,-0.0,-0.0,-0.0,-0.0,-1.0,-0.0,-0.0,-0.0,0.555673663731469,
        -0.027034185307057625,-0.70226225634217321,-0.027566488177000262,-0.7025340602672151,-0.026662833272981429,
        0.027034185307057625,0.027566488177000258,0.026662833272981429,0.0,0.0,0.0,0.0,1.0,0.0,0.0,0.0,0.0,-0.0,
        -0.0,-0.0,-0.0,-1.0,-0.0,-0.0,-0.0,0.026771909379554291,-0.55566424910285672,-0.62488504774223075,
        -0.024399835479656965,-0.63798948327222038,-0.021960985394712317,0.55566424910285672,0.62488504774223075,
        0.63798948327222038,0.0,0.0,0.0,0.0,1.0,0.0,0.0,0.0,0.0,-0.0,-0.0,-0.0,-0.0,-1.0,-0.0,-0.0,-0.0,
        0.62490021645747618,0.02706527731251647,0.026700746627905073,0.58505858013174894,-0.37854052611351124,
        -0.027072082181883242,-0.027610578309122807,-0.026708907388227909,0.027610578309122804,0.0,0.0,0.0,0.0,1.0,
        0.0,0.0,0.0,0.0,-0.0,-0.0,-0.0,-0.0,-1.0,-0.0,-0.0,0.027265477962947069,0.55566222109490582,
        0.63798667601923609,0.029437135799321903,-0.55566181651356428,-0.023469887537635181,-0.62488169574462793,
        -0.63798609648432814,0.0,0.0,0.0,0.0,1.0,0.0,0.0,0.0,0.0,-0.0,-0.0,-0.0,-0.0,-1.0,-0.0,-0.0,
        0.63800507768378822,-0.45692709004827581,-0.027011667529779945,-0.58505858013174894,-0.027541181508898387,
        -0.026637267215644224,0.027011667529779945,0.027541181508898383,0.026637267215644224,0.0,0.0,0.0,0.0,1.0,
        0.0,0.0,0.0,0.0,-0.0,-0.0,-0.0,-0.0,-1.0,-0.0,-0.0,0.026352061912650541,-0.55566389422834717,
        -0.02598312883534095,-0.62488507878410182,-0.02943713579932191,-0.637989575133729,0.55566389422834717,
        0.62488507878410182,0.63798957513372911,0.0,0.0,0.0,0.0,1.0,0.0,0.0,0.0,0.0,-0.0,-0.0,-0.0,-0.0,-1.0,-0.0,
        -0.0,-0.555673663731469,-0.027034185307057625,-0.027566488177000262,-0.026662833272981429,
        0.027034185307057625,0.70226225634217321,0.027566488177000258,0.7025340602672151,0.026662833272981429,0.0,
        0.0,0.0,0.0,1.0,0.0,0.0,0.0,0.0,-0.0,-0.0,-0.0,-0.0,-1.0,-0.0,-0.0,-0.0,-0.026771909379554291,
        -0.55566424910285672,-0.62488504774223075,-0.63798948327222038,0.55566424910285672,0.62488504774223075,
        0.024399835479656955,0.63798948327222038,0.021960985394712317,0.0,0.0,0.0,0.0,1.0,0.0,0.0,0.0,0.0,-0.0,-0.0,
        -0.0,-0.0,-1.0,-0.0,-0.0,-0.0,-0.62490021645747618,-0.58505858013174883,-0.027072082181883242,
        -0.027610578309122807,-0.026708907388227909,0.37854052611351124,0.027072082181883242,0.026708907388227909,
        0.0,0.0,0.0,0.0,1.0,0.0,0.0,0.0,-0.0,-0.0,-0.0,-0.0,-1.0,-0.0,-0.0,-0.0,-0.027265477962947069,
        -0.55566222109490582,-0.63798667601923609,-0.029437135799321879,-0.62488169574462793,0.55566181651356428,
        0.023469887537635192,0.62488169574462793,0.63798609648432814,0.0,0.0,0.0,0.0,1.0,0.0,0.0,0.0,-0.0,-0.0,-0.0,
        -0.0,-1.0,-0.0,-0.0,-0.0,-0.63800507768378822,-0.027011667529779945,-0.027541181508898387,
        -0.026637267215644224,0.45692709004827581,0.027011667529779945,0.58505858013174894,0.027541181508898383,
        0.026637267215644224,0.0,0.0,0.0,0.0,1.0,0.0,0.0,0.0,-0.0,-0.0,-0.0,-0.0,-1.0,-0.0,-0.0,-0.0,
        -0.026352061912650541,-0.55566389422834717,-0.62488507878410182,-0.637989575133729,0.55566389422834717,
        0.02598312883534095,0.62488507878410182,0.0294371357993219,0.63798957513372911,0.0,0.0,0.0,0.0,1.0,0.0,0.0,
        0.0,-0.0,-0.0,-0.0,-0.0,-1.0,-0.0,-0.0,-0.0,0.55566424910285672,0.027034185307057621,-0.70224208707170055,
        -0.024752136540096732,-0.70251617195999394,-0.022319435462106595,0.0,0.0,0.0,0.0,1.0,0.0,0.0,0.0,-0.0,-0.0,
        -0.0,-0.0,-1.0,-0.0,-0.0,-0.0,0.70226225634217332,0.3785405261135113,0.70163518723474272,
        -0.027105602758215112,-0.027648865450003536,-0.026748274296612785,0.027105602758215112,0.027648865450003533,
        0.026748274296612785,0.0,0.0,0.0,0.0,1.0,0.0,0.0,0.0,0.0,0.0,-0.0,-0.0,-0.0,-0.0,-1.0,-0.0,-0.0,
        0.55566222109490582,-0.023637206391576536,-0.015100165961297108,-0.0,0.378540460951947,0.02764886545000354,
        -0.015207454024849647,0.0,0.0,0.0,0.0,1.0,0.0,0.0,0.0,-0.0,-0.0,-0.0,-0.0,-1.0,-0.0,0.45692709004827575,
        0.702534060267215,-0.027090859530371859,-0.70163518723474272,0.026730661933064313,0.0,0.0,0.0,0.0,1.0,0.0,
        0.0,0.0,-0.0,-0.0,-0.0,-0.0,-1.0,-0.0,-0.0,0.55566389422834728,-0.029709944333287521,-0.0,
        0.37854017792555505,0.026748274296612796,0.0,0.0,0.0,0.0,1.0,0.0,0.0,0.0,0.0,-0.0,-0.0,-0.0,-0.0,-1.0,-0.0,
        0.55566424910285672,-0.027034185307057621,-0.0,0.37851997948504351,-0.70317323754735273,0.02240967789339866,
        0.0,0.0,0.0,0.0,1.0,0.0,0.0,0.0,-0.0,-0.0,-0.0,-0.0,-1.0,-0.0,-0.0,0.55566222109490582,
        -0.027566488177000255,-0.70223873149897853,0.023637206391576546,0.015100165961297143,0.0,0.0,0.0,1.0,0.0,
        0.0,-0.0,-0.0,-0.0,-0.0,-1.0,-0.0,-0.0,0.55566389422834728,-0.026662833272981429,-0.70224253943268344,
        -0.70251656286365771,0.026190122699982339,0.029709944333287511,0.0,0.0,0.0,0.0,1.0,0.0,0.0,-0.0,-0.0,-0.0,
        -0.0,-1.0,-0.0,-0.0,-0.0,0.02706527731251647,0.6248806237808493,0.023656120772106486,-0.378519539943052,
        -0.70317018870025627,0.0,0.0,0.0,0.0,1.0,0.0,0.0,0.0,-0.0,-0.0,-0.0,-0.0,-1.0,-0.0,0.02346980199155271,
        0.024399835479656976,-0.55566129015943833,-0.6248806237808493,-0.63798497169620461,-0.01473301981127613,
        0.55566129015943833,0.6248806237808493,0.63798497169620461,0.0,0.0,0.0,0.0,1.0,0.0,0.0,0.0,-0.0,-0.0,-0.0,
        -0.0,-1.0,-0.0,0.027011667529779945,0.63798948327222027,-0.456923837504278,-0.58504518410006956,
        -0.024723646828030479,0.0,0.0,0.0,0.0,1.0,0.0,0.0,0.0,-0.0,-0.0,-0.0,-0.0,-1.0,-0.0,-0.0,
        0.02598312883534095,0.021960985394712324,-0.63798532239475636,0.55566147407010114,0.62488096344828059,
        0.63798532239475636,0.0,0.0,0.0,0.0,1.0,0.0,0.0,0.0,0.0,0.0,-0.0,-0.0,-0.0,-0.0,-1.0,-0.0,-0.0,
        0.027034185307057618,-0.55566424910285683,-0.024752136540096732,0.70224208707170055,0.70251617195999394,0.0,
        0.0,0.0,0.0,1.0,0.0,0.0,0.0,-0.0,-0.0,-0.0,-0.0,-1.0,-0.0,-0.0,-0.0,0.02706527731251647,
        -0.62488504774223075,-0.024795740829694754,0.37851997948504357,0.7031738370963756,0.0,0.0,0.0,0.0,1.0,0.0,
        0.0,-0.0,-0.0,-0.0,-0.0,-1.0,-0.0,-0.0,0.027011667529779945,-0.63798948327222038,-0.024723646828030479,
        -0.02229166073122648,0.456923837504278,0.58504518410006945,0.0,0.0,0.0,0.0,1.0,0.0,0.0,-0.0,-0.0,-0.0,-0.0,
        -1.0,-0.0,-0.0,-0.0,0.6248822663250807,0.0276027315782233,0.58504257002809312,0.02974148887250478,
        -0.37854036201549385,-0.023660396850780661,0.0,0.0,0.0,0.0,1.0,0.0,0.0,0.0,-0.0,-0.0,-0.0,-0.0,-1.0,-0.0,
        0.62488507878410182,0.026700746627905073,0.58504502721143925,-0.37854017792555522,-0.029748443430697026,0.0,
        0.0,0.0,0.0,1.0,0.0,0.0,0.0,-0.0,-0.0,-0.0,-0.0,-1.0,-0.0,0.62488504774223086,0.022364818883998015,
        0.58504518410006956,-0.027072082181883231,-0.37854107343057747,0.024805000972806229,0.0,0.0,0.0,0.0,1.0,0.0,
        0.0,0.0,-0.0,-0.0,-0.0,-0.0,-1.0,-0.0,-0.0,0.58504257002809312,-0.027610578309122814,-0.37854046095194716,
        0.023660296965944735,0.015161281241640749,0.0,0.0,0.0,1.0,0.0,-0.0,-0.0,-0.0,-1.0,-0.0,0.027541181508898383,
        0.637986676019236,0.029685529684818829,-0.023621944154890266,-0.58504204394174086,0.0,0.0,0.0,0.0,1.0,0.0,
        0.0,0.0,-0.0,-0.0,-0.0,-0.0,-1.0,-0.0,0.027566488177000262,0.70251319697861081,0.029709944333287532,
        -0.55566181651356417,-0.023637304191565071,0.70223802681964376,0.0,0.0,0.0,0.0,1.0,0.0,0.0,0.0,-0.0,-0.0,
        -0.0,-0.0,-1.0,-0.0,-0.0,0.027602731578223291,0.02974148887250478,-0.62488169574462793,
        -0.023656120772106482,0.37851926782050033,0.70317150299940423,0.0,0.0,0.0,1.0,0.0,-0.0,-0.0,-0.0,-1.0,-0.0,
        0.027541181508898383,0.4569226479042604,0.58504257002809312,0.029685529684818829,-0.637986096484328,
        -0.023621944154890266,0.0,0.0,0.0,0.0,1.0,0.0,0.0,-0.0,-0.0,-0.0,-0.0,-1.0,-0.0,-0.0,0.637989575133729,
        0.026637267215644217,-0.58504502721143936,-0.029685529684818846,0.0,0.0,0.0,0.0,1.0,0.0,0.0,0.0,-0.0,-0.0,
        -0.0,-0.0,-1.0,-0.0,0.63798948327222038,-0.027011667529779945,-0.58504518410006945,0.024723646828030466,
        0.02229166073122648,0.0,0.0,0.0,0.0,1.0,0.0,0.0,0.0,-0.0,-0.0,-0.0,-0.0,-1.0,-0.0,-0.0,0.637986676019236,
        -0.02754118150889838,-0.58504257002809312,0.023621847095687702,0.015074517622588319,0.0,0.0,0.0,1.0,0.0,
        -0.0,-0.0,-0.0,-1.0,-0.0,0.637989575133729,-0.026637267215644217,-0.45692310525642205,-0.58504502721143936,
        0.026171339658097509,0.029685529684818822,0.0,0.0,0.0,0.0,1.0,0.0,0.0,-0.0,-0.0,-0.0,-0.0,-1.0,-0.0,-0.0,
        0.026662833272981426,-0.55566389422834728,-0.029709944333287525,0.70224253943268344,0.70251656286365771,0.0,
        0.0,0.0,0.0,1.0,0.0,0.0,0.0,-0.0,-0.0,-0.0,-0.0,-1.0,-0.0,-0.0,0.026700746627905069,-0.62488507878410182,
        -0.02974148887250477,0.37851908394641454,0.703174067452467,0.0,0.0,0.0,1.0,0.0,-0.0,-0.0,-0.0,-1.0,-0.0,
        0.026637267215644227,-0.637989575133729,-0.029685529684818811,0.456923105256422,0.58504502721143925,0.0,0.0,
        0.0,0.0,1.0,0.0,0.0,-0.0,-0.0,-0.0,-0.0,-1.0,-0.0,-0.0,-0.55566424910285672,-0.027034185307057621,
        0.70224208707170055,0.024752136540096722,0.70251617195999394,0.022319435462106609,0.0,0.0,0.0,0.0,1.0,0.0,
        0.0,0.0,-0.0,-0.0,-0.0,-0.0,-1.0,-0.0,-0.0,-0.0,-0.37851943317454484,-0.70226225634217332,
        -0.027098793108292794,0.70318478827029374,0.02674010789169564,0.0,0.0,0.0,0.0,1.0,0.0,0.0,-0.0,-0.0,-0.0,
        -0.0,-1.0,-0.0,-0.0,-0.0,-0.55566222109490582,-0.027566488177000255,0.023637206391576546,
        0.70223873149897853,0.70251319697861081,0.015100165961297143,0.0,0.0,0.0,1.0,0.0,-0.0,-0.0,-0.0,-1.0,-0.0,
        -0.0,-0.45692709004827575,-0.7025340602672151,-0.37854052611351124,-0.70318478827029385,
        -0.027105602758215112,-0.027648865450003536,-0.026748274296612785,0.027105602758215112,0.026748274296612785,
        0.0,0.0,0.0,0.0,1.0,0.0,0.0,0.0,-0.0,-0.0,-0.0,-0.0,-1.0,-0.0,-0.0,-0.0,-0.0,-0.55566389422834728,
        -0.026662833272981429,0.026190122699982339,0.70224253943268344,0.029709944333287511,0.70251656286365771,0.0,
        0.0,0.0,0.0,1.0,0.0,0.0,-0.0,-0.0,-0.0,-0.0,-1.0,-0.0,-0.0,-0.0,-0.02706527731251647,-0.62488504774223075,
        0.37851997948504357,0.024795740829694744,0.7031738370963756,0.022364818883998022,0.0,0.0,0.0,1.0,0.0,-0.0,
        -0.0,-0.0,-1.0,-0.0,-0.0,-0.02346980199155272,-0.024399835479656965,-0.55566129015943833,
        -0.6248806237808493,-0.63798497169620461,0.55566129015943833,0.6248806237808493,0.63798497169620461,
        0.014733019811276159,0.0,0.0,0.0,1.0,0.0,0.0,-0.0,-0.0,-0.0,-0.0,-1.0,-0.0,-0.0,-0.0,-0.027011667529779945,
        -0.63798948327222038,0.456923837504278,0.58504518410006945,0.024723646828030469,0.02229166073122648,0.0,0.0,
        0.0,0.0,1.0,0.0,0.0,-0.0,-0.0,-0.0,-0.0,-1.0,-0.0,-0.0,-0.0,-0.02598312883534095,-0.021960985394712324,
        -0.63798532239475636,0.55566147407010114,0.029307880059563592,0.0,0.0,0.0,0.0,1.0,0.0,0.0,-0.0,-0.0,-0.0,
        -0.0,-1.0,-0.0,-0.0,-0.6248822663250807,-0.027602731578223294,0.37851936679972537,0.023656021236335204,
        0.703171917764931,0.01515082442675411,0.0,0.0,1.0,0.0,-0.0,-0.0,-1.0,-0.0,-0.62488507878410182,
        -0.58504502721143936,-0.026708907388227905,0.37854017792555511,0.026218970645527549,0.029748443430697016,
        0.0,0.0,0.0,0.0,1.0,0.0,-0.0,-0.0,-0.0,-0.0,-1.0,-0.0,-0.0,-0.0,-0.02754118150889838,-0.63798667601923609,
        0.4569226479042604,0.023621847095687692,0.585042570028093,0.015074517622588279,0.0,0.0,0.0,0.0,1.0,0.0,-0.0,
        -0.0,-0.0,-0.0,-1.0,-0.0,-0.0,-0.63798957513372911,-0.026637267215644217,0.456923105256422,
        0.026171339658097509,0.58504502721143925,0.029685529684818822,0.0,0.0,0.0,0.0,1.0,0.0,-0.0,-0.0,-0.0,-0.0,
        -1.0,-0.0,-0.0,-0.0,0.702236447861886,0.37854073327939103,0.023682030674840704,0.00016424244292451563,
        -0.015216927320390218,0.0,0.0,0.0,0.0,1.0,0.0,0.0,0.0,0.0,-0.0,-0.0,-0.0,-0.0,-1.0,-0.0,0.55566129015943833,
        0.023637206391576532,0.024752136540096732,-0.702236447861886,-0.015109647396991065,0.0,0.0,0.0,0.0,1.0,0.0,
        -0.0,-0.0,-0.0,-1.0,-0.0,-0.0,0.45692383750427795,0.70251617195999394,0.37854107343057741,
        0.027105602758215115,-0.024849423695496659,0.0,0.0,0.0,0.0,1.0,0.0,0.0,0.0,0.0,-0.0,-0.0,-0.0,-0.0,-1.0,
        -0.0,-0.0,0.55566181651356428,-0.023637304191565081,-0.0,0.015196990314225767,0.37854036201549374,
        0.00027130052193601533,3.3862997711630647E-5,0.0,0.0,0.0,0.0,1.0,0.0,0.0,0.0,0.0,-0.0,-0.0,-0.0,-0.0,-1.0,
        -0.0,0.45692310525642194,0.70251656286365771,0.37854017792555505,0.70317346814293025,-0.026748274296612796,
        0.026245744732980112,0.029783569798323813,0.0,0.0,0.0,0.0,1.0,0.0,0.0,0.0,-0.0,-0.0,-0.0,-0.0,-1.0,-0.0,
        -0.0,0.55566129015943833,-0.023637206391576536,-0.024752136540096725,-0.702236447861886,
        0.015109647396991065,0.0,0.0,0.0,1.0,0.0,0.0,-0.0,-0.0,-0.0,-0.0,-1.0,-0.0,-0.0,-0.0,0.55566181651356428,
        -0.029709944333287493,-0.70223802681964376,-0.7025125679269647,0.023637304191565092,0.0,0.0,0.0,0.0,1.0,0.0,
        0.0,-0.0,-0.0,-0.0,-0.0,-1.0,-0.0,-0.0,-0.0,0.027072082181883235,0.58504518410006945,0.70317383709637549,
        -0.37854107343057752,-0.024805000972806222,0.0,0.0,0.0,0.0,1.0,0.0,0.0,0.0,-0.0,-0.0,-0.0,-0.0,-1.0,-0.0,
        -0.0,0.024723646828030497,0.63798497169620449,0.023621944154890263,-0.5850406398453023,0.0,0.0,0.0,0.0,1.0,
        0.0,0.0,0.0,0.0,-0.0,-0.0,-0.0,-0.0,-1.0,-0.0,0.023469887537635181,3.2815184442066549E-5,
        -0.55566088508118927,-0.62488005247477207,-0.63798439140804353,0.55566088508118927,0.62488005247477207,
        0.63798439140804353,0.0,0.0,0.0,0.0,1.0,0.0,0.0,0.0,0.0,0.0,-0.0,-0.0,-0.0,-0.0,-1.0,-0.0,-0.0,
        0.024752136540096736,0.70251116957088389,0.023637304191565078,-0.55566088508118927,0.7022357422084774,0.0,
        0.0,0.0,0.0,1.0,0.0,0.0,0.0,0.0,-0.0,-0.0,-0.0,-0.0,-1.0,-0.0,-0.0,0.024795740829694764,
        0.023656120772106475,-0.624880052474772,0.37851953994305221,0.70317018870025627,0.0,0.0,0.0,1.0,0.0,0.0,
        -0.0,-0.0,-0.0,-1.0,-0.0,0.023621847095687688,0.024723646828030497,-0.63798497169620461,
        -0.015083998191321592,0.45692247149286119,0.58504116656491612,0.0,0.0,0.0,0.0,1.0,0.0,0.0,-0.0,-0.0,-0.0,
        -0.0,-1.0,-0.0,0.023621944154890259,3.3598535051162514E-5,-0.0050973150136454475,0.45692225021991206,
        0.58504063984530219,0.0,0.0,0.0,0.0,1.0,0.0,0.0,0.0,-0.0,-0.0,-0.0,-0.0,-1.0,-0.0,-0.0,0.027098793108292798,
        -0.37851997948504373,-0.70224208707170055,0.70317323754735284,0.0,0.0,0.0,0.0,1.0,0.0,0.0,-0.0,-0.0,-0.0,
        -0.0,-1.0,-0.0,-0.0,-0.0,0.027090859530371859,0.023672783354342114,-0.4569224714928613,-0.70251116957088389,
        -0.015195086849570095,0.70160323232532973,0.0,0.0,0.0,1.0,0.0,0.0,-0.0,-0.0,-0.0,-0.0,-1.0,-0.0,-0.0,
        0.027072082181883235,-0.58504518410006934,-0.024805000972806222,-0.022374380992921029,0.37854107343057752,
        0.0,0.0,0.0,0.0,1.0,0.0,0.0,-0.0,-0.0,-0.0,-0.0,-1.0,-0.0,-0.0,-0.0,0.58504502721143925,0.70317406745246691,
        -0.026708907388227905,-0.37854017792555522,0.026218970645527549,0.029748443430697016,0.0,0.0,0.0,0.0,1.0,
        0.0,0.0,-0.0,-0.0,-0.0,-0.0,-1.0,-0.0,-0.0,0.585041166564916,-0.023660296965944742,-0.024805000972806225,
        -0.37854073327939119,0.015170756558948674,0.0,0.0,0.0,1.0,0.0,-0.0,-0.0,-1.0,-0.0,-0.0,-0.0,
        0.62488169574462793,0.58504204394174075,-0.029748443430697009,-0.37854036201549396,0.023660396850780658,0.0,
        0.0,0.0,0.0,1.0,0.0,0.0,-0.0,-0.0,-0.0,-0.0,-1.0,-0.0,-0.0,0.027631856629547157,-0.4569226479042604,
        -0.70251319697861081,-0.023672783354342117,-0.015185611969090922,0.70160605506782658,0.0,0.0,0.0,1.0,0.0,
        -0.0,-0.0,-0.0,-0.0,-1.0,-0.0,-0.0,0.027610578309122811,0.02974844343069703,-0.58504204394174075,
        -0.023660396850780651,0.37854036201549374,0.0,0.0,0.0,0.0,1.0,0.0,0.0,-0.0,-0.0,-0.0,-0.0,-1.0,-0.0,-0.0,
        0.63798497169620449,-0.0236218470956877,-0.024723646828030469,-0.58504116656491612,0.015083998191321633,0.0,
        0.0,0.0,1.0,0.0,-0.0,-0.0,-1.0,-0.0,-0.0,-0.0,-0.026171339658097509,-0.022291660731226463,
        -0.58504146009743707,0.0050973150136454448,-0.023621944154890263,-0.45692225021991223,0.0,0.0,0.0,0.0,1.0,
        0.0,0.0,-0.0,-0.0,-0.0,-0.0,-1.0,-0.0,-0.0,-0.0,0.637986096484328,-0.029685529684818798,
        -0.45692242688405121,-0.58504204394174086,0.02362194415489029,0.0,0.0,0.0,0.0,1.0,0.0,0.0,-0.0,-0.0,-0.0,
        -0.0,-1.0,-0.0,-0.0,0.026730661933064309,-0.45692310525642194,-0.70251656286365771,-0.029768291394636794,
        0.70161080096520145,0.0,0.0,0.0,0.0,1.0,0.0,0.0,-0.0,-0.0,-0.0,-0.0,-1.0,-0.0,-0.0,0.026708907388227905,
        -0.58504502721143925,-0.029748443430697019,0.378540177925555,0.0,0.0,0.0,0.0,1.0,0.0,0.0,-0.0,-0.0,-0.0,
        -0.0,-1.0,-0.0,-0.0,-0.4569238375042779,-0.027090859530371863,-0.70251617195999394,-0.37854107343057747,
        0.024849423695496649,0.022419246501157553,0.0,0.0,0.0,0.0,1.0,0.0,0.0,-0.0,-0.0,-0.0,-0.0,-1.0,-0.0,-0.0,
        -0.0,-0.0,-0.55566147407010114,-0.026190122699982339,-0.0223194354621066,0.70223692196481524,
        0.029647784654081327,0.70251158235928435,0.0,0.0,0.0,1.0,0.0,0.0,-0.0,-0.0,-0.0,-0.0,-1.0,-0.0,-0.0,-0.0,
        -0.70224253943268344,-0.378540177925555,-0.70161080096520145,-0.026748274296612796,0.029783569798323813,0.0,
        0.0,0.0,0.0,1.0,0.0,-0.0,-0.0,-0.0,-0.0,-1.0,-0.0,-0.0,-0.0,-0.0,-0.45692264790426035,-0.027631856629547154,
        -0.70251319697861092,0.023672783354342128,0.70160605506782658,0.015185611969090976,0.0,0.0,1.0,0.0,-0.0,
        -0.0,-0.0,-1.0,-0.0,-0.0,-0.55566181651356428,-0.029709944333287493,0.023637304191565092,
        0.70223802681964376,0.7025125679269647,0.0,0.0,0.0,0.0,1.0,0.0,0.0,-0.0,-0.0,-0.0,-0.0,-1.0,-0.0,-0.0,-0.0,
        -0.45692310525642188,-0.70251656286365771,-0.026730661933064316,0.026234238763943405,0.70161080096520145,
        0.029768291394636756,0.0,0.0,0.0,1.0,0.0,-0.0,-0.0,-0.0,-0.0,-1.0,-0.0,-0.0,-0.027072082181883235,
        -0.58504518410006934,0.37854107343057752,0.024805000972806211,0.022374380992921029,0.0,0.0,0.0,0.0,1.0,0.0,
        0.0,-0.0,-0.0,-0.0,-0.0,-1.0,-0.0,-0.0,-0.0,-0.026213688698745,-0.62488096344828059,-0.022364818883998026,
        0.3785195589565879,0.029687807671632122,0.70317085483536168,0.0,0.0,1.0,0.0,-0.0,-0.0,-0.0,-1.0,-0.0,-0.0,
        -0.023469887537635188,-0.00012845955535528616,-0.55566088508118927,-0.62488005247477207,
        -0.63798439140804353,0.55566088508118927,0.62488005247477207,0.63798439140804353,0.0,0.0,0.0,0.0,1.0,0.0,
        0.0,0.0,-0.0,-0.0,-0.0,-0.0,-1.0,-0.0,-0.0,-0.0,-0.0,-0.585042570028093,-0.027610578309122811,
        0.37854046095194716,0.023660296965944742,0.015161281241640751,0.0,0.0,0.0,0.0,1.0,0.0,-0.0,-0.0,-0.0,-0.0,
        -1.0,-0.0,-0.0,-0.62488169574462793,-0.029741488872504766,0.3785192678205006,0.023656120772106493,
        0.70317150299940423,0.0,0.0,0.0,0.0,1.0,0.0,-0.0,-0.0,-0.0,-0.0,-1.0,-0.0,-0.0,-0.029685529684818805,
        -0.637986096484328,0.45692242688405116,0.02362194415489028,0.58504204394174075,0.0,0.0,0.0,0.0,1.0,0.0,-0.0,
        -0.0,-0.0,-0.0,-1.0,-0.0,-0.0,-0.0,0.55566088508118927,0.023637304191565081,0.015109647396991093,
        -0.7022357422084774,0.0,0.0,0.0,0.0,1.0,0.0,0.0,0.0,0.0,-0.0,-0.0,-0.0,-0.0,-1.0,-0.0,-0.0,
        0.37854107343057741,0.0015613656062954475,-0.027105602758215108,0.02484942369549667,0.02241924650115756,0.0,
        0.0,0.0,0.0,1.0,0.0,0.0,0.0,0.0,-0.0,-0.0,-0.0,-0.0,-1.0,-0.0,-0.0,0.37854046095194693,0.70317131702755065,
        -0.027648865450003536,0.023682030674840704,0.015207454024849647,0.0,0.0,0.0,1.0,0.0,0.0,-0.0,-0.0,-0.0,-1.0,
        -0.0,0.702236447861886,-0.024840157186683216,0.37854073327939092,-0.023682030674840707,
        -0.0001642424429245156,0.015216927320390209,0.0,0.0,0.0,1.0,0.0,-0.0,-0.0,-1.0,-0.0,-0.0,-0.0,
        0.45692242688405105,0.7025125679269647,-0.02976829139463676,0.37854036201549374,-0.00027130052193601533,
        0.023682132033406258,0.0,0.0,0.0,0.0,1.0,0.0,0.0,0.0,-0.0,-0.0,-0.0,-0.0,-1.0,-0.0,-0.0,0.55566088508118927,
        -0.023637304191565085,-0.029647784654081352,-0.7022357422084774,-0.70251053960656562,0.0,0.0,0.0,0.0,1.0,
        0.0,0.0,-0.0,-0.0,-0.0,-0.0,-1.0,-0.0,-0.0,-0.0,-0.0,0.37851926782050049,0.70223802681964376,
        -0.029776610295742294,-0.70317090201170729,0.023677852874347757,0.0,0.0,0.0,0.0,1.0,0.0,0.0,-0.0,-0.0,-0.0,
        -0.0,-1.0,-0.0,0.58504116656491612,0.024805000972806236,0.70317060420331423,0.023660396850780658,
        0.0015608627398630522,-0.3785406342380947,0.0,0.0,0.0,0.0,1.0,0.0,0.0,0.0,0.0,-0.0,-0.0,-0.0,-0.0,-1.0,-0.0,
        0.023660296965944735,0.024805000972806239,-0.58504116656491578,-0.015170756558948695,0.37854073327939125,
        0.0,0.0,0.0,0.0,1.0,0.0,0.0,-0.0,-0.0,-0.0,-0.0,-1.0,-0.0,3.3895386058154954E-5,0.0,-0.0,
        0.023682030674840707,-0.37854073327939108,-0.0030612231608958297,0.0,0.0,0.0,0.0,1.0,0.0,0.0,-0.0,-0.0,-0.0,
        -0.0,-1.0,-0.0,-0.0,0.023660396850780651,3.37922497221569E-5,-0.0053104157804372727,0.37854063423809481,0.0,
        0.0,0.0,0.0,1.0,0.0,0.0,0.0,-0.0,-0.0,-0.0,-0.0,-1.0,-0.0,-0.0,0.027105602758215112,-0.37854107343057758,
        -0.0030612088654606811,-0.024849423695496673,-0.02241924650115756,0.0,0.0,0.0,0.0,1.0,0.0,0.0,-0.0,-0.0,
        -0.0,-0.0,-1.0,-0.0,-0.0,-0.0,-0.0,-0.026218970645527546,-0.022374380992921033,-0.37854065319208563,
        0.00531041578043727,-0.023660396850780661,0.0,0.0,0.0,0.0,1.0,0.0,0.0,-0.0,-0.0,-0.0,-0.0,-1.0,-0.0,-0.0,
        -0.0,0.015185611969090872,-0.45692242688405116,-0.7025125679269647,-0.023672883991351843,
        0.00027130052193601566,3.3862997711630437E-5,-0.3785403620154939,0.0,0.0,0.0,0.0,1.0,0.0,0.0,-0.0,-0.0,-0.0,
        -0.0,-1.0,-0.0,-0.0,-0.0,0.027648865450003536,-0.378540460951947,-0.70160605506782647,-0.0236820306748407,
        -0.015207454024849618,0.0,0.0,0.0,0.0,1.0,0.0,-0.0,-0.0,-0.0,-0.0,-1.0,-0.0,-0.0,-0.0,0.026748274296612789,
        -0.37854017792555505,-0.70161080096520156,-0.029783569798323847,0.0,0.0,0.0,0.0,1.0,0.0,0.0,-0.0,-0.0,-0.0,
        -0.0,-1.0,-0.0,-0.0,-0.0,-0.45692249061308471,-0.026234238763943405,-0.70251158235928435,
        -0.022398709579893369,0.70160383989347,0.029720779304182428,0.0,0.0,1.0,0.0,-0.0,-0.0,-0.0,-0.0,-1.0,-0.0,
        -0.0,-0.0,-0.55566088508118927,-0.023637304191565085,-0.029647784654081352,0.7022357422084774,
        0.70251053960656573,0.0,0.0,0.0,0.0,1.0,0.0,0.0,-0.0,-0.0,-0.0,-0.0,-1.0,-0.0,-0.0,-0.0,-0.0,
        -0.027648865450003536,-0.0,-0.37851926782050049,-0.70223802681964376,-0.029776610295742294,
        0.023677852874347757,0.0,0.0,0.0,0.0,1.0,0.0,-0.0,-0.0,-0.0,-0.0,-1.0,-0.0,-0.0,-0.0,-0.45692242688405105,
        -0.02976829139463676,-0.7025125679269647,0.023672883991351864,0.70160519311325342,0.0,0.0,0.0,1.0,0.0,-0.0,
        -0.0,-0.0,-0.0,-1.0,-0.0,-0.0,-0.62488005247477207,-0.023660396850780661,-0.0053104157804372719,
        -3.3792249722156905E-5,0.3785406342380947,0.0,0.0,0.0,0.0,1.0,0.0,-0.0,-0.0,-0.0,-0.0,-1.0,-0.0,-0.0,-0.0,
        -0.0,-0.023621944154890277,-0.00012982492179038625,-0.0050973150136454466,0.45692225021991212,
        0.5850406398453023,0.0,0.0,0.0,0.0,1.0,0.0,-0.0,-0.0,-0.0,-0.0,-1.0,-0.0,-0.0,-0.0,-0.0,
        -0.58504204394174064,-0.029748443430697026,-0.70317150299940412,-0.015161281241640776,0.37854036201549396,
        0.023660396850780654,0.0,0.0,0.0,0.0,1.0,0.0,-0.0,-0.0,-0.0,-0.0,-1.0,-0.0,-0.0,-0.0,0.378519539943052,
        0.023677852874347757,0.0046218484590718626,3.3872049431451388E-5,-0.70316958685172248,0.0,0.0,0.0,0.0,1.0,
        0.0,0.0,0.0,0.0,-0.0,-0.0,-0.0,-0.0,-1.0,-0.0,0.37854065319208546,-9.9046128627942282E-5,
        0.029739987791949973,0.0,0.0,0.0,1.0,0.0,0.0,0.0,0.0,0.0,-0.0,-0.0,-0.0,-0.0,-1.0,-0.0,-0.0,
        0.37851953994305204,-0.00013032533543202578,0.0030612242404972137,-0.023682132033406265,
        -0.00013036341924922685,0.0,0.0,0.0,0.0,1.0,0.0,0.0,0.0,-0.0,-0.0,-0.0,-0.0,-1.0,-0.0,-0.0,-0.0,
        0.45692225021991212,0.0030912635403395824,-0.02367288399135186,-0.70160236926968877,0.0,0.0,0.0,0.0,1.0,0.0,
        0.0,-0.0,-0.0,-0.0,-0.0,-1.0,-0.0,-0.0,-0.0,-0.45692225021991212,-0.02367288399135186,
        -0.00013027879750649216,-0.003091263540339582,0.70160236926968877,0.0,0.0,0.0,1.0,0.0,-0.0,-0.0,-0.0,-0.0,
        -1.0,-0.0,-0.0,-0.0,-0.378519539943052,-0.0046218484590718626,-0.023682132033406265,-3.389538605815513E-5,
        0.0,0.0,0.0,0.0,1.0,0.0,-0.0,-0.0,-0.0,-0.0,-1.0,-0.0,-0.0,-0.0,-0.0,-0.0,0.37854063423809459,
        0.023682132033406265,0.001561372566461268,3.389538605815513E-5,0.0,0.0,0.0,0.0,1.0,0.0,0.0,0.0,0.0,0.0,-0.0,
        -0.0,-0.0,-0.0,-1.0,-0.0,-0.047678521358187322,-0.55787204405389446,-0.048825402242851326,
        -0.62654723292970194,-0.047286920841764508,-0.63943141348019983,0.047678521358187322,0.55787204405389446,
        0.048825402242851333,0.62654723292970194,0.047286920841764508,0.63943141348019983,0.0,0.0,0.0,0.0,0.0,1.0,
        0.0,0.0,0.0,0.0,-0.0,-0.0,-0.0,-0.0,-0.0,-1.0,-0.0,-0.0,0.047678521358187315,-0.557872509055183,
        -0.044288901125137163,-0.62654217515979649,-0.040021361425923357,-0.63942545184526778,0.557872509055183,
        0.62654217515979649,0.63942545184526778,0.0,0.0,0.0,0.0,0.0,1.0,0.0,0.0,0.0,-0.0,-0.0,-0.0,-0.0,-0.0,-1.0,
        -0.0,-0.0,0.55787204405389446,-0.047942655141777091,-0.049117799127055072,-0.702875228655225,
        -0.0475823178492932,-0.70295568967385469,0.047942655141777091,0.049117799127055078,0.04758231784929319,0.0,
        0.0,0.0,0.0,0.0,1.0,0.0,0.0,0.0,-0.0,-0.0,-0.0,-0.0,-0.0,-1.0,-0.0,-0.0,0.048825402242851333,
        0.55787171658183987,0.63942424475811355,0.052452304750527382,-0.041298149353625656,-0.557871608027596,
        -0.62654080641868248,-0.63942401877909183,0.62654080641868248,0.0,0.0,0.0,0.0,0.0,1.0,0.0,0.0,0.0,-0.0,-0.0,
        -0.0,-0.0,-0.0,-1.0,-0.0,0.626547232929702,0.047984758880296075,0.04763006590676714,0.58732864799299578,
        -0.047993536136706469,-0.38140732638781982,-0.049174830154444668,-0.047640075741515714,0.0,0.0,0.0,0.0,0.0,
        1.0,0.0,0.0,0.0,-0.0,-0.0,-0.0,-0.0,-0.0,-1.0,-0.0,0.047286920841764508,-0.045941301434432633,
        -0.55787142569916037,-0.052452304750527444,-0.62654193427993921,-0.639425363845251,0.55787142569916037,
        0.62654193427993921,0.639425363845251,0.0,0.0,0.0,0.0,0.0,1.0,0.0,0.0,0.0,-0.0,-0.0,-0.0,-0.0,-0.0,-1.0,
        -0.0,0.63943141348019983,-0.047934264404490834,-0.45972838564453733,-0.0491093915715111,
        -0.58732864799299578,-0.04757405784581345,0.047934264404490834,0.0491093915715111,0.04757405784581345,0.0,
        0.0,0.0,0.0,0.0,1.0,0.0,0.0,0.0,-0.0,-0.0,-0.0,-0.0,-0.0,-1.0,-0.0,-0.047678521358187315,-0.557872509055183,
        -0.62654217515979649,-0.63942545184526778,0.557872509055183,0.044288901125137184,0.62654217515979649,
        0.04002136142592335,0.63942545184526778,0.0,0.0,0.0,0.0,0.0,1.0,0.0,0.0,0.0,-0.0,-0.0,-0.0,-0.0,-0.0,-1.0,
        -0.0,-0.0,-0.55787204405389446,-0.047942655141777091,-0.049117799127055072,-0.0475823178492932,
        0.047942655141777091,0.049117799127055078,0.702875228655225,0.04758231784929319,0.70295568967385469,0.0,0.0,
        0.0,0.0,0.0,1.0,0.0,0.0,0.0,-0.0,-0.0,-0.0,-0.0,-0.0,-1.0,-0.0,-0.0,-0.048825402242851333,
        -0.05245230475052743,-0.557871608027596,-0.62654080641868248,-0.63942401877909183,0.041298149353625628,
        0.557871608027596,0.63942401877909183,0.0,0.0,0.0,0.0,0.0,1.0,0.0,0.0,-0.0,-0.0,-0.0,-0.0,-0.0,-1.0,-0.0,
        -0.0,-0.626547232929702,-0.047984758880296075,-0.047630065906767147,-0.58732864799299578,
        -0.049174830154444668,0.047993536136706469,0.38140732638781982,0.049174830154444675,0.047640075741515707,
        0.0,0.0,0.0,0.0,0.0,1.0,0.0,0.0,-0.0,-0.0,-0.0,-0.0,-0.0,-1.0,-0.0,-0.0,-0.047286920841764508,
        -0.55787142569916037,-0.62654193427993921,-0.639425363845251,0.045941301434432633,0.55787142569916037,
        0.052452304750527472,0.62654193427993921,0.639425363845251,0.0,0.0,0.0,0.0,0.0,1.0,0.0,0.0,-0.0,-0.0,-0.0,
        -0.0,-0.0,-1.0,-0.0,-0.0,-0.63943141348019983,-0.047934264404490834,-0.0491093915715111,
        -0.04757405784581345,0.047934264404490834,0.45972838564453733,0.0491093915715111,0.58732864799299578,
        0.04757405784581345,0.0,0.0,0.0,0.0,0.0,1.0,0.0,0.0,-0.0,-0.0,-0.0,-0.0,-0.0,-1.0,-0.0,-0.0,
        0.047942655141777091,0.557872509055183,-0.044607913288060984,-0.70286297549379462,-0.040334527208629158,
        -0.70294446596883164,0.0,0.0,0.0,0.0,0.0,1.0,0.0,0.0,-0.0,-0.0,-0.0,-0.0,-0.0,-1.0,-0.0,-0.0,
        0.04428890112513717,0.041298149353625621,0.052879406986409215,-0.557871950150472,-0.62654033525020214,
        -0.6394234093758725,0.557871950150472,0.62654033525020214,0.6394234093758725,0.0,0.0,0.0,0.0,0.0,1.0,0.0,
        0.0,0.0,0.0,-0.0,-0.0,-0.0,-0.0,-0.0,-1.0,-0.0,0.047984758880296068,-0.38139322558672084,
        -0.70313339581753054,-0.0,0.041515729018567704,0.62654033525020214,-0.70313108620605158,0.0,0.0,0.0,0.0,0.0,
        1.0,0.0,0.0,-0.0,-0.0,-0.0,-0.0,-0.0,-1.0,0.045941301434432633,0.040021361425923357,-0.55787198584888142,
        -0.0528794069864092,0.63942378652894072,0.0,0.0,0.0,0.0,0.0,1.0,0.0,0.0,-0.0,-0.0,-0.0,-0.0,-0.0,-1.0,-0.0,
        0.047934264404490841,-0.587326232489261,-0.0,0.041479097778282452,0.6394234093758725,0.0,0.0,0.0,0.0,0.0,
        1.0,0.0,0.0,0.0,-0.0,-0.0,-0.0,-0.0,-0.0,-1.0,0.047942655141777091,-0.557872509055183,-0.0,
        0.041486488318378048,-0.027677161979573293,0.70294159791647837,0.0,0.0,0.0,0.0,0.0,1.0,0.0,0.0,-0.0,-0.0,
        -0.0,-0.0,-0.0,-1.0,-0.0,0.047984758880296068,-0.62654217515979649,-0.044660621016635559,
        0.38139322558672084,0.70313339581753065,0.0,0.0,0.0,0.0,1.0,0.0,-0.0,-0.0,-0.0,-0.0,-0.0,-1.0,-0.0,
        0.047934264404490841,-0.63942545184526778,-0.0446006835917423,-0.040327604063683457,0.45973364369000819,
        0.587326232489261,0.0,0.0,0.0,0.0,0.0,1.0,0.0,-0.0,-0.0,-0.0,-0.0,-0.0,-1.0,-0.0,-0.0,0.55787171658183987,
        0.049198241144151271,0.38141432182325924,-0.041543427917705961,-0.027753531302003462,0.0,0.0,0.0,0.0,0.0,
        1.0,0.0,0.0,-0.0,-0.0,-0.0,-0.0,-0.0,-1.0,0.381386025829566,0.702875228655225,-0.048014979218259819,
        -0.049198241144151264,-0.047663646280299156,-0.70314122138856006,0.048014979218259819,0.049198241144151271,
        0.047663646280299156,0.0,0.0,0.0,0.0,0.0,1.0,0.0,0.0,-0.0,-0.0,-0.0,-0.0,-0.0,-1.0,0.55787142569916048,
        0.04758231784929319,-0.046165728248822986,-0.052734339992385214,-0.70286396678410767,0.0,0.0,0.0,0.0,0.0,
        1.0,0.0,0.0,-0.0,-0.0,-0.0,-0.0,-0.0,-1.0,-0.0,0.45972838564453744,0.70295568967385458,-0.04765651814247162,
        0.048008393947647693,0.049191105586226781,0.047656518142471613,0.0,0.0,0.0,0.0,0.0,1.0,0.0,0.0,0.0,0.0,-0.0,
        -0.0,-0.0,-0.0,-0.0,-1.0,-0.0,0.557872509055183,-0.0479426551417771,-0.70286297549379462,
        0.044607913288061025,0.040334527208629151,0.0,0.0,0.0,0.0,0.0,1.0,0.0,0.0,-0.0,-0.0,-0.0,-0.0,-0.0,-1.0,
        -0.0,-0.0,0.55787171658183987,-0.049117799127055085,-0.70286143698134129,0.041486488318378041,
        0.027661054311066195,0.0,0.0,0.0,0.0,0.0,1.0,0.0,-0.0,-0.0,-0.0,-0.0,-0.0,-1.0,-0.0,0.55787142569916048,
        -0.04758231784929319,-0.70286396678410767,-0.70294533564091966,0.046165728248822986,0.052734339992385255,
        0.0,0.0,0.0,0.0,0.0,1.0,0.0,-0.0,-0.0,-0.0,-0.0,-0.0,-1.0,-0.0,-0.0,0.049164972356125373,
        0.62654101707515264,0.052779600708881172,0.58732523320298258,-0.041521734602731605,-0.38141436310945664,0.0,
        0.0,0.0,0.0,0.0,1.0,0.0,0.0,-0.0,-0.0,-0.0,-0.0,-0.0,-1.0,0.049109391571511091,0.63942424475811355,
        0.052725613098002319,-0.041479097778282452,-0.58732507052489791,0.0,0.0,0.0,0.0,0.0,1.0,0.0,0.0,-0.0,-0.0,
        -0.0,-0.0,-0.0,-1.0,0.049117799127055078,0.70294302173702006,0.052734339992385228,-0.557871608027596,
        -0.041486711482857687,0.70286111061272671,0.0,0.0,0.0,0.0,0.0,1.0,0.0,0.0,-0.0,-0.0,-0.0,-0.0,-0.0,-1.0,
        -0.0,0.052779600708881172,-0.62654080641868259,-0.041515729018567711,0.381393060579516,0.70313207851881332,
        0.0,0.0,0.0,0.0,1.0,-0.0,-0.0,-0.0,-0.0,-1.0,0.62654193427993921,0.047630065906767147,0.58732556690019289,
        -0.38141260703668056,-0.052788975072809517,0.0,0.0,0.0,0.0,0.0,1.0,0.0,0.0,-0.0,-0.0,-0.0,-0.0,-0.0,-1.0,
        0.62654217515979649,0.040386220026432475,0.587326232489261,-0.047993536136706476,-0.38141452789755637,
        0.044671688889686353,0.0,0.0,0.0,0.0,0.0,1.0,0.0,0.0,-0.0,-0.0,-0.0,-0.0,-0.0,-1.0,-0.0,0.62654101707515253,
        0.58732523320298247,-0.049174830154444668,-0.38141432182325907,0.041521509739207062,0.027720209169872088,
        0.0,0.0,0.0,0.0,1.0,-0.0,-0.0,-0.0,-0.0,-1.0,0.62654193427993921,0.04620090230449761,0.0527796007088812,
        0.58732556690019289,-0.0476400757415157,-0.38141260703668056,0.0,0.0,0.0,0.0,0.0,1.0,0.0,-0.0,-0.0,-0.0,
        -0.0,-0.0,-1.0,-0.0,0.047574057845813457,0.639425363845251,-0.052725613098002347,-0.58732556690019289,0.0,
        0.0,0.0,0.0,0.0,1.0,0.0,0.0,-0.0,-0.0,-0.0,-0.0,-0.0,-1.0,0.04758231784929319,-0.55787142569916037,
        -0.052734339992385269,0.70286396678410767,0.70294533564091966,0.0,0.0,0.0,0.0,0.0,1.0,0.0,0.0,-0.0,-0.0,
        -0.0,-0.0,-0.0,-1.0,-0.0,0.04763006590676714,-0.62654193427993921,-0.052779600708881193,0.38139130491870232,
        0.703133933677141,0.0,0.0,0.0,0.0,1.0,-0.0,-0.0,-0.0,-0.0,-1.0,0.047574057845813457,-0.639425363845251,
        -0.04615757913241255,-0.052725613098002347,0.45973190050489804,0.58732556690019289,0.0,0.0,0.0,0.0,0.0,1.0,
        0.0,-0.0,-0.0,-0.0,-0.0,-0.0,-1.0,-0.0,0.63942545184526778,-0.047934264404490834,-0.587326232489261,
        0.044600683591742338,0.04032760406368343,0.0,0.0,0.0,0.0,0.0,1.0,0.0,0.0,-0.0,-0.0,-0.0,-0.0,-0.0,-1.0,-0.0,
        0.63942424475811355,-0.0491093915715111,-0.58732523320298258,0.041478874690674995,0.027655051949837254,0.0,
        0.0,0.0,0.0,1.0,-0.0,-0.0,-0.0,-0.0,-1.0,0.639425363845251,-0.047574057845813443,-0.58732556690019289,
        0.04615757913241255,0.052725613098002382,0.0,0.0,0.0,0.0,0.0,1.0,0.0,-0.0,-0.0,-0.0,-0.0,-0.0,-1.0,-0.0,
        -0.047942655141777091,-0.557872509055183,0.044607913288061012,0.70286297549379462,0.040334527208629144,
        0.70294446596883164,0.0,0.0,0.0,0.0,0.0,1.0,0.0,0.0,-0.0,-0.0,-0.0,-0.0,-0.0,-1.0,-0.0,-0.0,
        -0.041297934356687133,-0.0442889011251372,-0.55787205898156167,0.027381569976781938,0.63942363589545237,0.0,
        0.0,0.0,0.0,0.0,1.0,0.0,-0.0,-0.0,-0.0,-0.0,-0.0,-1.0,-0.0,-0.0,-0.047984758880296068,-0.62654217515979649,
        0.38139322558672084,0.044660621016635579,0.040386220026432489,0.70313339581753065,0.0,0.0,0.0,0.0,1.0,-0.0,
        -0.0,-0.0,-0.0,-1.0,-0.0,-0.045941301434432633,-0.04002136142592335,-0.041298149353625628,
        -0.027381569976781941,-0.557871950150472,-0.62654033525020214,-0.6394234093758725,0.557871950150472,
        0.6394234093758725,0.0,0.0,0.0,0.0,0.0,1.0,0.0,0.0,-0.0,-0.0,-0.0,-0.0,-0.0,-1.0,-0.0,-0.0,-0.0,
        -0.047934264404490841,-0.63942545184526778,0.45973364369000819,0.044600683591742324,0.587326232489261,
        0.040327604063683443,0.0,0.0,0.0,0.0,0.0,1.0,0.0,-0.0,-0.0,-0.0,-0.0,-0.0,-1.0,-0.0,-0.0,
        -0.55787171658183987,-0.049117799127055085,0.041486488318378041,0.70286143698134129,0.027661054311066195,
        0.70294302173702006,0.0,0.0,0.0,0.0,1.0,-0.0,-0.0,-0.0,-0.0,-1.0,-0.0,-0.381386025829566,
        -0.70287522865522511,-0.048014979218259819,-0.049198241144151264,-0.047663646280299156,0.048014979218259819,
        0.049198241144151271,0.047663646280299156,0.70314122138856006,0.0,0.0,0.0,0.0,1.0,0.0,-0.0,-0.0,-0.0,-0.0,
        -0.0,-1.0,-0.0,-0.0,-0.55787142569916048,-0.04758231784929319,0.046165728248822986,0.052734339992385255,
        0.70286396678410767,0.70294533564091966,0.0,0.0,0.0,0.0,0.0,1.0,0.0,-0.0,-0.0,-0.0,-0.0,-0.0,-1.0,-0.0,-0.0,
        -0.45972838564453744,-0.70295568967385458,-0.04765651814247162,0.048008393947647693,0.70268597089371387,0.0,
        0.0,0.0,0.0,0.0,1.0,0.0,-0.0,-0.0,-0.0,-0.0,-0.0,-1.0,-0.0,-0.049164972356125373,-0.62654101707515264,
        0.041515504461835731,0.38139301933175634,0.027709698583410016,0.70313230364575241,0.0,0.0,0.0,1.0,-0.0,-0.0,
        -0.0,-1.0,-0.049109391571511105,-0.052725613098002361,-0.63942401877909172,0.041479097778282459,
        0.45973321032477427,0.58732507052489791,0.0,0.0,0.0,0.0,0.0,1.0,-0.0,-0.0,-0.0,-0.0,-0.0,-1.0,-0.0,-0.0,
        -0.62654193427993921,-0.047630065906767147,0.04620090230449761,0.38139130491870232,0.052779600708881227,
        0.703133933677141,0.0,0.0,0.0,0.0,0.0,1.0,-0.0,-0.0,-0.0,-0.0,-0.0,-1.0,-0.0,-0.047574057845813457,
        -0.639425363845251,0.046157579132412557,0.45973190050489804,0.052725613098002388,0.58732556690019289,0.0,
        0.0,0.0,0.0,0.0,1.0,-0.0,-0.0,-0.0,-0.0,-0.0,-1.0,-0.0,-0.0,0.044696511233766632,0.041537644408465073,
        0.38139435220779871,0.0046455551781967915,-0.70313098732427648,0.0,0.0,0.0,0.0,0.0,1.0,0.0,0.0,0.0,-0.0,
        -0.0,-0.0,-0.0,-0.0,-1.0,0.048014979218259812,0.38139322558672073,0.70286297549379451,-0.04469651123376666,
        -0.70313329820348291,0.0,0.0,0.0,0.0,0.0,1.0,-0.0,-0.0,-0.0,-0.0,-1.0,-0.0,0.046165728248822986,
        0.040334527208629165,0.041486711482857673,0.55787195015047186,-0.70285954634074388,0.0,0.0,0.0,0.0,0.0,1.0,
        0.0,0.0,0.0,-0.0,-0.0,-0.0,-0.0,-0.0,-1.0,-0.0,0.047993536136706476,-0.38141452789755642,-0.0,
        0.70313131216765046,0.0415217346027316,0.0053499825507371153,0.0015656878741349531,0.0,0.0,0.0,0.0,0.0,1.0,
        0.0,0.0,0.0,-0.0,-0.0,-0.0,-0.0,-0.0,-1.0,0.04615757913241255,0.040327604063683457,0.041479097778282452,
        0.027671157031094271,-0.6394234093758725,0.45973424542066693,0.58732499879699229,0.0,0.0,0.0,0.0,0.0,1.0,
        0.0,0.0,-0.0,-0.0,-0.0,-0.0,-0.0,-1.0,-0.0,0.048014979218259812,-0.38139322558672073,-0.70286297549379451,
        -0.04469651123376666,0.70313329820348291,0.0,0.0,0.0,0.0,1.0,0.0,-0.0,-0.0,-0.0,-0.0,-0.0,-1.0,-0.0,-0.0,
        0.047993536136706476,-0.587326232489261,-0.044671688889686333,-0.040397149349959804,0.38141452789755642,0.0,
        0.0,0.0,0.0,0.0,1.0,0.0,-0.0,-0.0,-0.0,-0.0,-0.0,-1.0,-0.0,-0.0,0.557871608027596,0.052734339992385235,
        0.027661054311066337,-0.041486711482857694,-0.70286111061272671,0.0,0.0,0.0,0.0,0.0,1.0,0.0,0.0,-0.0,-0.0,
        -0.0,-0.0,-0.0,-1.0,-0.0,0.70286396678410779,0.047663646280299149,0.38141260703668067,-0.052821149416567043,
        0.0,0.0,0.0,0.0,0.0,1.0,0.0,0.0,0.0,-0.0,-0.0,-0.0,-0.0,-0.0,-1.0,0.38140732638781988,0.0015661221639725058,
        -0.048023761687426413,-0.049208104725552843,-0.047673661972528605,0.048023761687426413,0.049208104725552849,
        0.0476736619725286,0.0,0.0,0.0,0.0,0.0,1.0,0.0,0.0,0.0,0.0,-0.0,-0.0,-0.0,-0.0,-0.0,-1.0,-0.0,
        0.70286297549379451,0.04042146861842183,0.38141452789755653,-0.048023761687426413,0.044707585477670696,0.0,
        0.0,0.0,0.0,0.0,1.0,0.0,0.0,0.0,-0.0,-0.0,-0.0,-0.0,-0.0,-1.0,-0.0,0.70286143698134129,0.38141432182325918,
        -0.049208104725552843,0.041543427917705954,0.027753531302003361,0.0,0.0,0.0,0.0,1.0,0.0,-0.0,-0.0,-0.0,-0.0,
        -1.0,0.38139130491870249,0.70286396678410779,-0.047663646280299149,-0.70313383642924188,
        0.046226776721425993,0.052811769511494744,0.0,0.0,0.0,0.0,0.0,1.0,0.0,-0.0,-0.0,-0.0,-0.0,-0.0,-1.0,
        0.38141260703668073,0.0015661807001885121,-0.0003808990881292652,0.046234063364270737,0.052821149416567105,
        0.0,0.0,0.0,0.0,0.0,1.0,0.0,0.0,-0.0,-0.0,-0.0,-0.0,-0.0,-1.0,-0.0,0.55787205898156167,
        -0.041486488318378034,-0.044607913288061032,0.02767716197957313,0.0,0.0,0.0,0.0,0.0,1.0,0.0,-0.0,-0.0,-0.0,
        -0.0,-0.0,-1.0,-0.0,-0.0,0.55787198584888142,0.38139402411953655,-0.046226776721426013,-0.04042146861842183,
        -0.70313145912642394,0.053301939043787668,0.0,0.0,0.0,0.0,1.0,0.0,-0.0,-0.0,-0.0,-0.0,-0.0,-1.0,-0.0,
        0.557871608027596,-0.052734339992385269,-0.70286111061272671,-0.70294271779415229,0.041486711482857687,0.0,
        0.0,0.0,0.0,0.0,1.0,0.0,-0.0,-0.0,-0.0,-0.0,-0.0,-1.0,-0.0,-0.0,0.052725613098002319,0.027655051949837452,
        -0.63942401877909172,-0.041479097778282452,0.45973321032477427,0.58732507052489791,0.0,0.0,0.0,0.0,0.0,1.0,
        0.0,-0.0,-0.0,-0.0,-0.0,-0.0,-1.0,-0.0,0.052811769511494709,-0.381393060579516,-0.70286111061272671,
        -0.041537644408465066,0.70313198021515855,0.0,0.0,0.0,0.0,1.0,-0.0,-0.0,-0.0,-1.0,-0.0,-0.0,
        0.049174830154444661,0.052788975072809545,-0.58732507052489813,-0.041521734602731612,0.38141436310945631,
        0.0,0.0,0.0,0.0,0.0,1.0,0.0,-0.0,-0.0,-0.0,-0.0,-0.0,-1.0,-0.0,0.6265406645097189,-0.046200902304497617,
        -0.040386220026432475,-0.38139402411953627,-0.70313155774868141,0.053264773578912634,0.0,0.0,0.0,0.0,1.0,
        -0.0,-0.0,-0.0,-0.0,-0.0,-1.0,-0.0,0.62654080641868248,0.58732507052489791,-0.052788975072809559,
        -0.38141436310945637,0.0415217346027316,0.0,0.0,0.0,0.0,0.0,1.0,0.0,-0.0,-0.0,-0.0,-0.0,-0.0,-1.0,-0.0,
        0.047663646280299156,-0.38139130491870238,-0.70286396678410779,-0.052811769511494681,0.70313383642924188,
        0.0,0.0,0.0,0.0,1.0,-0.0,-0.0,-0.0,-1.0,-0.0,-0.0,-0.45973190050489809,-0.70294533564091954,
        -0.052804674695198853,0.00038089908812926509,-0.38141260703668056,-0.046234063364270724,0.0,0.0,0.0,0.0,0.0,
        1.0,0.0,-0.0,-0.0,-0.0,-0.0,-0.0,-1.0,-0.0,-0.0,0.047640075741515714,-0.58732556690019289,
        -0.046208184541143907,-0.0527889750728095,0.38141260703668045,0.0,0.0,0.0,0.0,0.0,1.0,0.0,-0.0,-0.0,-0.0,
        -0.0,-0.0,-1.0,-0.0,0.63942378652894072,-0.046157579132412543,-0.040327604063683443,-0.587325187651558,
        0.053202204406742878,0.0,0.0,0.0,0.0,0.0,1.0,0.0,-0.0,-0.0,-0.0,-0.0,-0.0,-1.0,-0.0,0.63942401877909172,
        -0.052725613098002388,-0.5873250705248978,0.041479097778282417,0.0,0.0,0.0,0.0,0.0,1.0,0.0,-0.0,-0.0,-0.0,
        -0.0,-0.0,-1.0,-0.0,-0.046165728248822993,-0.55787198584888142,-0.040334527208629144,-0.041486711482857666,
        0.70285954634074388,0.70294129315678422,0.0,0.0,0.0,0.0,0.0,1.0,0.0,-0.0,-0.0,-0.0,-0.0,-0.0,-1.0,-0.0,-0.0,
        -0.0,-0.048008393947647693,-0.45973364369000813,-0.70294446596883153,0.04468906953870326,0.7026717750678485,
        0.040414301735567953,0.0,0.0,0.0,0.0,1.0,0.0,-0.0,-0.0,-0.0,-0.0,-0.0,-1.0,-0.0,-0.0,-0.044600683591742331,
        -0.041479097778282431,-0.053202204406742781,-0.6394234093758725,0.58732499879699229,0.0,0.0,0.0,0.0,0.0,1.0,
        -0.0,-0.0,-0.0,-0.0,-0.0,-1.0,-0.0,-0.0,-0.0,-0.04620090230449761,-0.62654066450971879,
        -0.040386220026432489,0.38139402411953638,0.053264773578912634,0.70313155774868152,0.0,0.0,0.0,1.0,-0.0,
        -0.0,-0.0,-0.0,-1.0,-0.0,-0.047993536136706476,-0.587326232489261,0.38141452789755642,0.044671688889686353,
        0.040397149349959791,0.0,0.0,0.0,0.0,0.0,1.0,0.0,-0.0,-0.0,-0.0,-0.0,-0.0,-1.0,-0.0,-0.0,
        -0.046157579132412557,-0.040327604063683437,-0.63942378652894072,0.4597340245185435,0.0532022044067428,
        0.58732518765155828,0.0,0.0,0.0,0.0,1.0,-0.0,-0.0,-0.0,-0.0,-0.0,-1.0,-0.0,-0.557871608027596,
        -0.052734339992385269,0.041486711482857687,0.70286111061272671,0.70294271779415229,0.0,0.0,0.0,0.0,0.0,1.0,
        0.0,-0.0,-0.0,-0.0,-0.0,-0.0,-1.0,-0.0,-0.0,-0.45973321958975349,-0.049191105586226788,-0.70294302173702006,
        0.041532433509010709,0.70267008402296527,0.027736669979992645,0.0,0.0,0.0,1.0,-0.0,-0.0,-0.0,-0.0,-1.0,-0.0,
        -0.38140732638781988,-0.0030799473449444718,-0.048023761687426413,-0.049208104725552843,
        -0.047673661972528605,0.048023761687426413,0.049208104725552849,0.0476736619725286,0.0,0.0,0.0,0.0,0.0,1.0,
        0.0,0.0,-0.0,-0.0,-0.0,-0.0,-0.0,-1.0,-0.0,-0.0,-0.0,-0.052779600708881207,-0.62654080641868259,
        0.0415157290185677,0.38139306057951583,0.70313207851881332,0.0,0.0,0.0,0.0,0.0,1.0,-0.0,-0.0,-0.0,-0.0,-0.0,
        -1.0,-0.0,-0.049174830154444675,-0.58732523320298258,0.041521509739207041,0.381414321823259,
        0.027720209169872008,0.0,0.0,0.0,0.0,0.0,1.0,-0.0,-0.0,-0.0,-0.0,-0.0,-1.0,-0.0,-0.58732556690019289,
        -0.047640075741515707,0.046208184541143907,0.38141260703668056,0.052788975072809566,0.0,0.0,0.0,0.0,0.0,1.0,
        -0.0,-0.0,-0.0,-0.0,-0.0,-1.0,-0.0,-0.0,0.048023761687426413,0.38141452789755642,0.70313329820348291,
        -0.044707585477670654,0.0,0.0,0.0,0.0,0.0,1.0,0.0,0.0,0.0,-0.0,-0.0,-0.0,-0.0,-0.0,-1.0,-0.0,
        0.0414867114828577,6.14559350203706E-5,-0.55787195015047186,0.70285954634074388,0.70294129315678422,0.0,0.0,
        0.0,0.0,0.0,1.0,0.0,0.0,0.0,-0.0,-0.0,-0.0,-0.0,-0.0,-1.0,-0.0,0.041515729018567704,0.027725808084743217,
        -0.62654033525020214,0.38139435220779894,0.70313108620605158,0.0,0.0,0.0,0.0,1.0,0.0,-0.0,-0.0,-0.0,-0.0,
        -1.0,0.044696511233766639,-0.70285987351907608,0.04153764440846508,-0.3813943522077986,
        -0.0046455551781967924,0.70313098732427659,0.0,0.0,0.0,0.0,1.0,-0.0,-0.0,-0.0,-1.0,-0.0,-0.0,
        0.046208184541143921,0.040397149349959804,-0.58732518765155828,0.041521734602731619,-0.0053499825507371188,
        0.38141565496819624,0.0,0.0,0.0,0.0,0.0,1.0,0.0,0.0,-0.0,-0.0,-0.0,-0.0,-0.0,-1.0,-0.0,0.048023761687426413,
        -0.38141452789755642,-0.7026717750678485,-0.044707585477670654,-0.040432404230908,0.0,0.0,0.0,0.0,0.0,1.0,
        0.0,-0.0,-0.0,-0.0,-0.0,-0.0,-1.0,-0.0,-0.0,-0.0,0.041521509739207062,0.044671688889686333,
        -0.58732516183395489,-0.027736318903840668,0.3814156136550157,0.0,0.0,0.0,0.0,0.0,1.0,0.0,-0.0,-0.0,-0.0,
        -0.0,-0.0,-1.0,0.052811769511494695,0.70286111061272671,0.027743014678389594,0.38141436310945653,
        6.1605929268691053E-5,-0.04154365368638769,0.0,0.0,0.0,0.0,0.0,1.0,0.0,0.0,0.0,-0.0,-0.0,-0.0,-0.0,-0.0,
        -1.0,0.38139306057951616,0.70286111061272671,-0.052811769511494744,-0.70313198021515855,0.04153764440846508,
        0.0,0.0,0.0,0.0,0.0,1.0,0.0,-0.0,-0.0,-0.0,-0.0,-0.0,-1.0,0.0015662095088587794,0.0,-0.0,
        0.38139435220779888,-0.041537644408465059,-0.00023256610403676135,0.0,0.0,0.0,0.0,0.0,1.0,0.0,-0.0,-0.0,
        -0.0,-0.0,-0.0,-1.0,-0.0,0.38141436310945653,0.0015661981899676553,-0.0004794577441265344,
        0.041543653686387648,0.0,0.0,0.0,0.0,0.0,1.0,0.0,0.0,-0.0,-0.0,-0.0,-0.0,-0.0,-1.0,-0.0,0.55787195015047186,
        -0.041486711482857659,-0.00023216176133703439,-0.70285954634074388,-0.70294129315678422,0.0,0.0,0.0,0.0,0.0,
        1.0,0.0,-0.0,-0.0,-0.0,-0.0,-0.0,-1.0,-0.0,-0.0,-0.0,-0.45973321032477421,-0.70294271779415229,
        -0.041532658817056131,0.0004794577441265338,-0.38141436310945637,0.0,0.0,0.0,0.0,0.0,1.0,0.0,-0.0,-0.0,-0.0,
        -0.0,-0.0,-1.0,-0.0,-0.0,0.70313155774868141,-0.046208184541143935,-0.040397149349959777,
        -0.38141532678103607,0.0053499825507371248,0.0015656878741349477,-0.041521734602731612,0.0,0.0,0.0,0.0,0.0,
        1.0,0.0,-0.0,-0.0,-0.0,-0.0,-0.0,-1.0,-0.0,-0.0,0.62654033525020214,-0.041515729018567704,
        -0.053264773578912579,-0.38139435220779877,-0.70313108620605158,0.0,0.0,0.0,0.0,0.0,1.0,-0.0,-0.0,-0.0,-0.0,
        -0.0,-1.0,-0.0,-0.0,0.63942340937587239,-0.041479097778282424,-0.053202204406742795,-0.58732499879699218,
        0.0,0.0,0.0,0.0,0.0,1.0,0.0,-0.0,-0.0,-0.0,-0.0,-0.0,-1.0,-0.0,-0.0,-0.046220967236855211,
        -0.45973402451854339,-0.04041430173556794,-0.7029419471796341,0.05329394831239747,0.70266869475347082,0.0,
        0.0,0.0,1.0,-0.0,-0.0,-0.0,-0.0,-0.0,-1.0,-0.0,-0.0,-0.048023761687426413,-0.38141452789755642,
        -0.7026717750678485,0.044707585477670675,0.040432404230907985,0.0,0.0,0.0,0.0,0.0,1.0,0.0,-0.0,-0.0,-0.0,
        -0.0,-0.0,-1.0,-0.0,-0.0,-0.0,-0.62654033525020214,-0.0,-0.041521509739207055,-0.04467168888968636,
        -0.58732516183395489,0.3814156136550157,0.0,0.0,0.0,0.0,0.0,1.0,-0.0,-0.0,-0.0,-0.0,-0.0,-1.0,-0.0,-0.0,
        -0.046208184541143914,-0.58732518765155806,-0.040397149349959791,0.38141532678103618,0.053276115903559441,
        0.0,0.0,0.0,0.0,1.0,-0.0,-0.0,-0.0,-0.0,-0.0,-1.0,-0.0,-0.049208104725552843,-0.38141436310945653,
        -0.00047945774412653418,-0.0015661981899676573,0.041543653686387676,0.0,0.0,0.0,0.0,0.0,1.0,-0.0,-0.0,-0.0,
        -0.0,-0.0,-1.0,-0.0,-0.0,-0.0,-0.38141260703668067,-0.0030800493725469838,-0.00038089908812926525,
        0.046234063364270724,0.052821149416567063,0.0,0.0,0.0,0.0,0.0,1.0,-0.0,-0.0,-0.0,-0.0,-0.0,-1.0,-0.0,-0.0,
        -0.0,-0.052788975072809573,-0.5873250705248978,-0.027720209169872036,-0.70313207851881321,
        0.041521734602731585,0.38141436310945664,0.0,0.0,0.0,0.0,0.0,1.0,-0.0,-0.0,-0.0,-0.0,-0.0,-1.0,-0.0,-0.0,
        0.041543427917705968,0.38141561365501536,0.00029424831666778297,0.0015662085872463908,-0.027769643467705708,
        0.0,0.0,0.0,0.0,0.0,1.0,0.0,0.0,0.0,-0.0,-0.0,-0.0,-0.0,-0.0,-1.0,0.041532658817056138,
        -0.0031055287133001592,0.70266788285587956,0.0,0.0,0.0,0.0,1.0,0.0,0.0,0.0,0.0,-0.0,-0.0,-0.0,-0.0,-0.0,
        -1.0,-0.0,0.041543427917705961,-0.0030801002245625041,0.00023261598934981646,-0.381415654968196,
        -0.0030801017285724173,0.0,0.0,0.0,0.0,0.0,1.0,0.0,0.0,-0.0,-0.0,-0.0,-0.0,-0.0,-1.0,-0.0,-0.0,
        0.046234063364270724,0.00017791507742684638,-0.38141532678103585,-0.053313287899267439,0.0,0.0,0.0,0.0,0.0,
        1.0,0.0,-0.0,-0.0,-0.0,-0.0,-0.0,-1.0,-0.0,-0.0,-0.04623406336427073,-0.38141532678103612,
        -0.003080095298344224,-0.00017791507742684627,0.053313287899267488,0.0,0.0,0.0,0.0,1.0,-0.0,-0.0,-0.0,-0.0,
        -0.0,-1.0,-0.0,-0.0,-0.041543427917705961,-0.00029424831666778313,-0.38141565496819613,
        -0.0015662095088587807,0.0,0.0,0.0,0.0,0.0,1.0,-0.0,-0.0,-0.0,-0.0,-0.0,-1.0,-0.0,-0.0,-0.0,-0.0,
        0.041543653686387669,0.38141565496819613,6.1661881147355389E-5,0.0015662095088587807,0.0,0.0,0.0,0.0,0.0,
        1.0,0.0,0.0,0.0,0.0,-0.0,-0.0,-0.0,-0.0,-0.0,-1.0,0.555673663731469,0.026771909379554294,
        0.62490021645747618,0.027265477962947069,0.63800507768378811,0.026352061912650541,-0.555673663731469,
        -0.026771909379554294,-0.62490021645747618,-0.027265477962947066,-0.63800507768378822,-0.026352061912650541,
        0.0,0.0,0.0,0.0,0.0,0.0,1.0,0.0,0.0,0.0,-0.0,-0.0,-0.0,-0.0,-0.0,-0.0,-1.0,-0.0,-0.555673663731469,
        0.027034185307057625,0.70226225634217321,0.027566488177000262,0.7025340602672151,0.026662833272981429,
        -0.027034185307057625,-0.027566488177000258,-0.026662833272981429,0.0,0.0,0.0,0.0,0.0,0.0,0.0,0.0,0.0,-0.0,
        -0.0,-0.0,-0.0,-0.0,-0.0,-1.0,-0.0,-0.026771909379554291,0.55566424910285672,0.62488504774223075,
        0.024399835479656965,0.63798948327222038,0.021960985394712317,-0.55566424910285672,-0.62488504774223075,
        -0.63798948327222038,0.0,0.0,0.0,0.0,0.0,0.0,1.0,0.0,0.0,-0.0,-0.0,-0.0,-0.0,-0.0,-0.0,-1.0,-0.0,
        -0.62490021645747618,-0.02706527731251647,-0.026700746627905073,-0.58505858013174894,0.37854052611351124,
        0.027072082181883242,0.027610578309122807,0.026708907388227909,-0.027610578309122804,0.0,0.0,0.0,0.0,0.0,
        0.0,1.0,0.0,0.0,-0.0,-0.0,-0.0,-0.0,-0.0,-0.0,-0.0,-0.027265477962947069,-0.55566222109490582,
        -0.63798667601923609,-0.029437135799321903,0.55566181651356428,0.023469887537635181,0.62488169574462793,
        0.63798609648432814,0.0,0.0,0.0,0.0,0.0,0.0,1.0,0.0,0.0,-0.0,-0.0,-0.0,-0.0,-0.0,-0.0,-1.0,
        -0.63800507768378822,0.45692709004827581,0.027011667529779945,0.58505858013174894,0.027541181508898387,
        0.026637267215644224,-0.027011667529779945,-0.027541181508898383,-0.026637267215644224,0.0,0.0,0.0,0.0,0.0,
        0.0,1.0,0.0,0.0,-0.0,-0.0,-0.0,-0.0,-0.0,-0.0,-0.0,-0.026352061912650541,0.55566389422834717,
        0.02598312883534095,0.62488507878410182,0.02943713579932191,0.637989575133729,-0.55566389422834717,
        -0.62488507878410182,-0.63798957513372911,0.0,0.0,0.0,0.0,0.0,0.0,1.0,0.0,0.0,-0.0,-0.0,-0.0,-0.0,-0.0,-0.0,
        -1.0,0.555673663731469,0.027034185307057625,0.027566488177000262,0.026662833272981429,-0.027034185307057625,
        -0.70226225634217321,-0.027566488177000258,-0.7025340602672151,-0.026662833272981429,0.0,0.0,0.0,0.0,0.0,
        0.0,1.0,0.0,0.0,-0.0,-0.0,-0.0,-0.0,-0.0,-0.0,-0.0,-0.0,0.026771909379554291,0.55566424910285672,
        0.62488504774223075,0.63798948327222038,-0.55566424910285672,-0.62488504774223075,-0.024399835479656955,
